Yaskawa INFORM job: DPRINT3D3.JBI

/JOB
//NAME DPRINT3D3
//POS
///NPOS 1003,0,0,0,0,0
///TOOL 9
///POSTYPE PULSE
///PULSE
C00000=29899,52059,-123343,60719,-118918,-94818,0
C00001=29890,52052,-123365,60727,-118907,-94823,0
C00002=29880,52046,-123386,60735,-118894,-94827,0
C00003=29870,52040,-123408,60743,-118882,-94832,0
C00004=29861,52034,-123430,60750,-118870,-94837,0
C00005=29851,52028,-123450,60758,-118858,-94842,0
C00006=29842,52022,-123472,60766,-118846,-94847,0
C00007=29832,52016,-123494,60774,-118834,-94852,0
C00008=29824,52011,-123510,60781,-118825,-94855,0
C00009=29816,52006,-123527,60788,-118815,-94859,0
C00010=29807,52001,-123543,60795,-118805,-94863,0
C00011=29799,51997,-123561,60802,-118795,-94866,0
C00012=29789,51992,-123577,60810,-118786,-94870,0
C00013=29780,51988,-123593,60818,-118777,-94872,0
C00014=29772,51983,-123609,60825,-118766,-94876,0
C00015=29762,51978,-123626,60833,-118757,-94879,0
C00016=29753,51974,-123642,60841,-118747,-94883,0
C00017=29744,51969,-123658,60849,-118738,-94886,0
C00018=29735,51964,-123674,60857,-118727,-94890,0
C00019=29726,51960,-123691,60865,-118718,-94893,0
C00020=29717,51955,-123707,60872,-118709,-94897,0
C00021=29708,51951,-123724,60880,-118699,-94900,0
C00022=29699,51946,-123740,60888,-118689,-94904,0
C00023=29690,51941,-123756,60896,-118680,-94907,0
C00024=29682,51937,-123770,60903,-118671,-94910,0
C00025=29674,51934,-123782,60911,-118663,-94912,0
C00026=29665,51930,-123796,60918,-118655,-94915,0
C00027=29657,51926,-123810,60926,-118647,-94918,0
C00028=29649,51922,-123824,60933,-118638,-94921,0
C00029=29640,51918,-123836,60941,-118630,-94924,0
C00030=29632,51915,-123850,60948,-118622,-94926,0
C00031=29624,51911,-123862,60956,-118614,-94929,0
C00032=29615,51908,-123874,60964,-118607,-94931,0
C00033=29611,51906,-123881,60968,-118602,-94932,0
C00034=29593,51903,-123889,60986,-118593,-94932,0
C00035=29559,51898,-123908,61022,-118574,-94933,0
C00036=29524,51893,-123925,61058,-118556,-94933,0
C00037=29489,51888,-123943,61094,-118537,-94934,0
C00038=29463,51884,-123955,61122,-118524,-94934,0
C00039=29436,51881,-123966,61150,-118510,-94933,0
C00040=29409,51878,-123977,61178,-118497,-94933,0
C00041=29384,51875,-123986,61204,-118486,-94932,0
C00042=29360,51873,-123994,61230,-118474,-94932,0
C00043=29335,51870,-124003,61256,-118463,-94931,0
C00044=29310,51868,-124011,61283,-118450,-94930,0
C00045=29285,51865,-124019,61309,-118439,-94929,0
C00046=29260,51863,-124028,61335,-118427,-94928,0
C00047=29238,51861,-124034,61359,-118418,-94928,0
C00048=29218,51859,-124040,61380,-118409,-94926,0
C00049=29198,51858,-124046,61402,-118401,-94925,0
C00050=29178,51856,-124050,61423,-118392,-94924,0
C00051=29158,51855,-124055,61445,-118384,-94923,0
C00052=29141,51853,-124059,61463,-118376,-94922,0
C00053=29134,51853,-124061,61471,-118373,-94921,0
C00054=29119,51858,-124043,61489,-118376,-94915,0
C00055=29105,51862,-124026,61506,-118378,-94908,0
C00056=29091,51867,-124010,61524,-118380,-94901,0
C00057=29077,51872,-123993,61542,-118383,-94894,0
C00058=29063,51876,-123975,61560,-118385,-94888,0
C00059=29049,51881,-123958,61577,-118387,-94881,0
C00060=29035,51886,-123941,61595,-118389,-94875,0
C00061=29021,51890,-123924,61613,-118392,-94868,0
C00062=29007,51895,-123907,61630,-118394,-94861,0
C00063=28992,51901,-123887,61650,-118397,-94853,0
C00064=28977,51906,-123866,61669,-118401,-94846,0
C00065=28962,51912,-123847,61688,-118404,-94838,0
C00066=28947,51917,-123826,61707,-118408,-94830,0
C00067=28931,51924,-123804,61727,-118411,-94822,0
C00068=28914,51931,-123779,61748,-118416,-94813,0
C00069=28898,51937,-123755,61770,-118420,-94803,0
C00070=28881,51944,-123730,61791,-118425,-94794,0
C00071=28865,51951,-123704,61813,-118430,-94785,0
C00072=28848,51958,-123680,61834,-118434,-94776,0
C00073=28832,51965,-123655,61855,-118439,-94766,0
C00074=28815,51972,-123631,61877,-118443,-94757,0
C00075=28799,51979,-123604,61898,-118449,-94748,0
C00076=28783,51987,-123578,61919,-118454,-94738,0
C00077=28767,51994,-123550,61940,-118460,-94728,0
C00078=28745,52005,-123510,61969,-118469,-94713,0
C00079=28723,52017,-123470,61999,-118478,-94699,0
C00080=28701,52028,-123428,62029,-118487,-94684,0
C00081=28679,52039,-123387,62058,-118496,-94670,0
C00082=28657,52051,-123347,62088,-118504,-94655,0
C00083=28633,52064,-123299,62120,-118517,-94639,0
C00084=28605,52082,-123237,62159,-118532,-94617,0
C00085=28573,52102,-123163,62204,-118550,-94592,0
C00086=28541,52123,-123088,62248,-118569,-94566,0
C00087=28512,52142,-123021,62289,-118587,-94543,0
C00088=28512,52148,-123000,62292,-118595,-94537,0
C00089=28511,52154,-122979,62295,-118603,-94531,0
C00090=28511,52160,-122960,62298,-118611,-94525,0
C00091=28511,52165,-122940,62300,-118618,-94520,0
C00092=28511,52171,-122918,62303,-118627,-94514,0
C00093=28512,52178,-122896,62305,-118637,-94507,0
C00094=28513,52185,-122872,62307,-118646,-94500,0
C00095=28514,52192,-122847,62310,-118656,-94494,0
C00096=28515,52199,-122823,62312,-118666,-94487,0
C00097=28515,52206,-122798,62314,-118677,-94480,0
C00098=28517,52213,-122773,62316,-118687,-94473,0
C00099=28518,52220,-122748,62318,-118697,-94466,0
C00100=28518,52227,-122724,62320,-118707,-94459,0
C00101=28519,52234,-122699,62322,-118717,-94452,0
C00102=28520,52241,-122675,62325,-118727,-94445,0
C00103=28521,52248,-122649,62327,-118738,-94438,0
C00104=28522,52255,-122624,62329,-118748,-94431,0
C00105=28544,52343,-122318,62346,-118877,-94346,0
C00106=28565,52431,-122013,62363,-119005,-94261,0
C00107=22726,60437,-97506,72380,-124352,-86432,0
C00108=22603,60494,-97345,72531,-124324,-86367,0
C00109=22480,60552,-97184,72683,-124295,-86302,0
C00110=22469,60557,-97168,72696,-124293,-86296,0
C00111=22459,60563,-97152,72710,-124290,-86289,0
C00112=22448,60569,-97136,72724,-124288,-86283,0
C00113=22437,60574,-97120,72737,-124286,-86277,0
C00114=22427,60580,-97104,72751,-124285,-86271,0
C00115=22416,60586,-97088,72764,-124282,-86264,0
C00116=22405,60591,-97072,72778,-124280,-86258,0
C00117=22394,60597,-97057,72791,-124278,-86252,0
C00118=22384,60603,-97041,72805,-124275,-86246,0
C00119=22373,60608,-97025,72818,-124273,-86239,0
C00120=22362,60614,-97009,72832,-124272,-86233,0
C00121=22352,60619,-96994,72844,-124270,-86227,0
C00122=22344,60625,-96980,72855,-124269,-86222,0
C00123=22335,60630,-96965,72866,-124267,-86217,0
C00124=22327,60635,-96951,72877,-124266,-86211,0
C00125=22318,60640,-96936,72888,-124265,-86206,0
C00126=22310,60645,-96921,72900,-124264,-86200,0
C00127=22302,60651,-96905,72911,-124263,-86194,0
C00128=22293,60657,-96890,72922,-124263,-86188,0
C00129=22285,60662,-96875,72933,-124262,-86182,0
C00130=22277,60668,-96859,72944,-124260,-86177,0
C00131=22268,60673,-96843,72955,-124259,-86171,0
C00132=22260,60679,-96828,72966,-124259,-86166,0
C00133=22251,60684,-96812,72977,-124258,-86160,0
C00134=22225,60745,-96644,73033,-124287,-86108,0
C00135=22211,60785,-96532,73066,-124309,-86074,0
C00136=22198,60827,-96416,73100,-124332,-86039,0
C00137=22185,60869,-96300,73134,-124354,-86004,0
C00138=22179,60891,-96239,73150,-124367,-85986,0
C00139=22173,60913,-96177,73167,-124380,-85967,0
C00140=22169,60935,-96117,73181,-124393,-85950,0
C00141=22165,60956,-96059,73196,-124406,-85932,0
C00142=22161,60977,-96000,73210,-124419,-85915,0
C00143=22157,60998,-95940,73225,-124432,-85897,0
C00144=22153,61020,-95881,73239,-124446,-85880,0
C00145=22150,61038,-95832,73250,-124457,-85866,0
C00146=22148,61055,-95783,73261,-124468,-85852,0
C00147=22145,61073,-95734,73272,-124480,-85837,0
C00148=22144,61089,-95691,73281,-124490,-85825,0
C00149=22143,61104,-95648,73290,-124501,-85813,0
C00150=22142,61120,-95605,73299,-124511,-85800,0
C00151=22141,61135,-95563,73307,-124521,-85788,0
C00152=22139,61151,-95520,73316,-124532,-85776,0
C00153=22138,61166,-95477,73325,-124543,-85763,0
C00154=22137,61182,-95434,73334,-124554,-85751,0
C00155=22137,61195,-95397,73340,-124563,-85740,0
C00156=22137,61209,-95359,73347,-124572,-85730,0
C00157=22136,61222,-95322,73354,-124582,-85719,0
C00158=22136,61236,-95285,73361,-124591,-85708,0
C00159=22136,61249,-95248,73368,-124601,-85698,0
C00160=22136,61261,-95215,73373,-124610,-85689,0
C00161=22137,61273,-95183,73378,-124619,-85679,0
C00162=22137,61285,-95150,73384,-124627,-85671,0
C00163=22138,61297,-95117,73389,-124636,-85661,0
C00164=22138,61309,-95085,73394,-124645,-85652,0
C00165=22139,61320,-95052,73400,-124653,-85643,0
C00166=22139,61332,-95019,73405,-124663,-85633,0
C00167=22139,61344,-94987,73411,-124672,-85624,0
C00168=22153,61355,-94956,73403,-124687,-85618,0
C00169=22165,61365,-94930,73395,-124702,-85613,0
C00170=22178,61374,-94904,73387,-124717,-85607,0
C00171=22190,61384,-94878,73379,-124730,-85602,0
C00172=22203,61394,-94852,73372,-124745,-85596,0
C00173=22215,61403,-94825,73364,-124759,-85591,0
C00174=22231,61414,-94797,73354,-124776,-85585,0
C00175=22246,61424,-94768,73344,-124794,-85580,0
C00176=22261,61435,-94739,73334,-124811,-85574,0
C00177=22277,61446,-94710,73324,-124827,-85568,0
C00178=22292,61456,-94681,73314,-124844,-85563,0
C00179=22307,61467,-94651,73304,-124861,-85557,0
C00180=22326,61479,-94619,73290,-124882,-85551,0
C00181=22345,61491,-94587,73278,-124902,-85545,0
C00182=22364,61502,-94554,73265,-124922,-85539,0
C00183=22388,61516,-94517,73248,-124947,-85532,0
C00184=22412,61529,-94481,73231,-124971,-85526,0
C00185=22421,61530,-94478,73222,-124976,-85527,0
C00186=22431,61531,-94476,73213,-124983,-85527,0
C00187=22440,61532,-94473,73204,-124989,-85528,0
C00188=22449,61533,-94470,73195,-124996,-85529,0
C00189=22458,61535,-94467,73187,-125002,-85530,0
C00190=22468,61535,-94465,73178,-125009,-85531,0
C00191=22477,61537,-94462,73169,-125015,-85531,0
C00192=22487,61537,-94460,73160,-125021,-85532,0
C00193=22497,61538,-94459,73150,-125028,-85534,0
C00194=22507,61539,-94457,73141,-125034,-85535,0
C00195=22517,61539,-94455,73131,-125041,-85536,0
C00196=22526,61540,-94453,73122,-125048,-85537,0
C00197=22536,61541,-94452,73112,-125055,-85538,0
C00198=38402,60566,-97394,77280,-121677,-85721,0
C00199=38418,60624,-97233,77289,-121724,-85676,0
C00200=38452,60740,-96909,77308,-121819,-85588,0
C00201=38470,60804,-96733,77318,-121870,-85539,0
C00202=38473,60814,-96704,77319,-121879,-85531,0
C00203=38477,60825,-96675,77320,-121887,-85524,0
C00204=38480,60835,-96646,77321,-121897,-85516,0
C00205=38484,60846,-96617,77322,-121906,-85508,0
C00206=38488,60856,-96588,77323,-121914,-85500,0
C00207=38491,60866,-96560,77324,-121923,-85492,0
C00208=38495,60877,-96531,77326,-121932,-85484,0
C00209=38498,60887,-96501,77327,-121941,-85476,0
C00210=38502,60898,-96473,77328,-121950,-85469,0
C00211=38505,60908,-96444,77329,-121959,-85461,0
C00212=38509,60919,-96415,77330,-121968,-85453,0
C00213=38512,60927,-96391,77330,-121975,-85447,0
C00214=38516,60936,-96368,77331,-121983,-85440,0
C00215=38519,60944,-96344,77331,-121990,-85434,0
C00216=38523,60953,-96320,77332,-121998,-85427,0
C00217=38527,60961,-96297,77331,-122006,-85421,0
C00218=38531,60970,-96273,77331,-122013,-85415,0
C00219=38534,60978,-96250,77331,-122021,-85409,0
C00220=38538,60987,-96226,77331,-122029,-85402,0
C00221=38542,60996,-96203,77331,-122037,-85396,0
C00222=38546,61004,-96179,77331,-122045,-85390,0
C00223=38550,61013,-96156,77331,-122053,-85384,0
C00224=38554,61021,-96132,77331,-122060,-85378,0
C00225=38556,61025,-96120,77330,-122064,-85375,0
C00226=38617,61064,-96014,77289,-122127,-85352,0
C00227=38658,61088,-95950,77259,-122166,-85340,0
C00228=38700,61111,-95887,77227,-122207,-85328,0
C00229=38743,61134,-95824,77196,-122248,-85315,0
C00230=38766,61145,-95793,77178,-122269,-85310,0
C00231=38789,61157,-95762,77161,-122291,-85304,0
C00232=38812,61166,-95736,77143,-122310,-85300,0
C00233=38834,61176,-95710,77125,-122330,-85295,0
C00234=38856,61185,-95684,77108,-122351,-85291,0
C00235=38879,61195,-95657,77090,-122370,-85286,0
C00236=38901,61205,-95631,77073,-122390,-85282,0
C00237=38920,61212,-95611,77058,-122406,-85279,0
C00238=38938,61219,-95592,77042,-122422,-85276,0
C00239=38957,61226,-95573,77027,-122438,-85273,0
C00240=38974,61232,-95557,77014,-122452,-85271,0
C00241=38990,61238,-95542,77000,-122466,-85270,0
C00242=39007,61243,-95527,76986,-122479,-85267,0
C00243=39024,61249,-95512,76972,-122493,-85266,0
C00244=39040,61254,-95497,76958,-122507,-85264,0
C00245=39057,61260,-95482,76945,-122521,-85261,0
C00246=39073,61265,-95467,76931,-122534,-85260,0
C00247=39088,61270,-95456,76918,-122546,-85259,0
C00248=39103,61274,-95445,76906,-122557,-85257,0
C00249=39117,61278,-95434,76894,-122570,-85256,0
C00250=39132,61282,-95422,76881,-122582,-85255,0
C00251=39146,61286,-95411,76869,-122593,-85254,0
C00252=39159,61289,-95403,76857,-122603,-85253,0
C00253=39172,61292,-95395,76846,-122613,-85253,0
C00254=39185,61296,-95386,76835,-122623,-85253,0
C00255=39198,61299,-95378,76824,-122633,-85252,0
C00256=39211,61302,-95370,76812,-122642,-85252,0
C00257=39224,61305,-95361,76801,-122653,-85251,0
C00258=39237,61308,-95353,76790,-122663,-85250,0
C00259=39250,61311,-95344,76779,-122672,-85250,0
C00260=39255,61309,-95352,76772,-122675,-85253,0
C00261=39266,61303,-95367,76760,-122677,-85259,0
C00262=39280,61295,-95389,76742,-122680,-85267,0
C00263=39293,61288,-95410,76725,-122684,-85275,0
C00264=39307,61280,-95432,76708,-122687,-85284,0
C00265=39321,61272,-95454,76691,-122691,-85292,0
C00266=39335,61264,-95476,76674,-122694,-85300,0
C00267=39351,61254,-95503,76654,-122698,-85310,0
C00268=39366,61244,-95531,76634,-122701,-85320,0
C00269=39382,61234,-95558,76614,-122705,-85331,0
C00270=39398,61225,-95586,76594,-122708,-85340,0
C00271=39414,61215,-95614,76574,-122711,-85351,0
C00272=39430,61205,-95641,76554,-122714,-85361,0
C00273=39448,61192,-95676,76530,-122717,-85374,0
C00274=39466,61180,-95711,76507,-122721,-85387,0
C00275=39484,61167,-95746,76483,-122723,-85400,0
C00276=39506,61151,-95791,76455,-122725,-85415,0
C00277=39527,61135,-95836,76427,-122728,-85432,0
C00278=39530,61127,-95858,76420,-122725,-85438,0
C00279=39534,61120,-95879,76413,-122723,-85444,0
C00280=39538,61112,-95899,76406,-122719,-85451,0
C00281=39542,61105,-95920,76398,-122717,-85458,0
C00282=39545,61097,-95941,76391,-122715,-85464,0
C00283=39549,61089,-95962,76384,-122711,-85471,0
C00284=39553,61082,-95983,76377,-122709,-85477,0
C00285=39556,61074,-96006,76370,-122706,-85484,0
C00286=39560,61066,-96028,76363,-122703,-85491,0
C00287=39563,61058,-96051,76356,-122700,-85498,0
C00288=39567,61050,-96073,76348,-122696,-85505,0
C00289=39571,61041,-96096,76341,-122693,-85512,0
C00290=39574,61033,-96118,76334,-122691,-85519,0
C00291=40253,57939,-104914,74266,-120876,-88158,0
C00292=39352,58001,-104714,75214,-120443,-87977,0
C00293=39289,57986,-104756,75273,-120398,-87981,0
C00294=38619,57932,-104903,75932,-119998,-87936,0
C00295=37942,57980,-104749,76638,-119667,-87804,0
C00296=37297,58130,-104299,77353,-119421,-87590,0
C00297=37222,58161,-104207,77441,-119401,-87554,0
C00298=36275,57663,-105643,78197,-118546,-87864,0
C00299=41043,57280,-106870,73160,-120764,-88836,0
C00300=41858,56647,-108775,72029,-120639,-89503,0
C00301=35258,57163,-107098,79033,-117663,-88181,0
C00302=34216,56686,-108501,79913,-116799,-88491,0
C00303=42701,56041,-110631,70871,-120503,-90160,0
C00304=43572,55460,-112438,69686,-120353,-90807,0
C00305=33148,56231,-109853,80834,-115950,-88792,0
C00306=32056,55798,-111153,81799,-115118,-89085,0
C00307=44472,54905,-114198,68471,-120191,-91442,0
C00308=45402,54374,-115911,67227,-120017,-92067,0
C00309=30938,55387,-112402,82805,-114303,-89372,0
C00310=30073,55089,-113315,83596,-113696,-89584,0
C00311=30084,55047,-113445,83573,-113676,-89626,0
C00312=30076,54952,-113743,83553,-113615,-89719,0
C00313=46130,53866,-117579,66205,-119735,-92649,0
C00314=46001,53590,-118484,66218,-119365,-92894,0
C00315=45984,53367,-119225,66135,-119095,-93108,0
C00316=25619,60155,-98330,69289,-125787,-87153,0
C00317=25520,59915,-99002,69267,-125531,-87324,0
C00318=25252,59544,-100046,69355,-125071,-87569,0
C00319=46086,52886,-120853,65807,-118548,-93596,0
C00320=46100,52846,-120989,65774,-118503,-93638,0
C00321=46138,52799,-121152,65710,-118458,-93690,0
C00322=45305,52415,-122459,66450,-117684,-93972,0
C00323=25512,58771,-102250,68697,-124545,-88230,0
C00324=26027,57961,-104598,67753,-124084,-88973,0
C00325=44250,51964,-124020,67407,-116754,-94317,0
C00326=36507,55621,-111785,55133,-126158,-92810,0
C00327=26561,57182,-106893,66801,-123611,-89703,0
C00328=27117,56433,-109139,65839,-123127,-90421,0
C00329=35436,55163,-113183,56093,-125149,-92963,0
C00330=34338,54728,-114530,57095,-124159,-93114,0
C00331=27695,55714,-111338,64867,-122633,-91128,0
C00332=28295,55023,-113491,63881,-122127,-91823,0
C00333=33211,54314,-115828,58137,-123193,-93261,0
C00334=32057,53921,-117076,59221,-122246,-93405,0
C00335=31078,54046,-116653,60363,-122047,-93134,0
C00336=31078,53985,-116676,60373,-122074,-93115,0
C00337=46650,54077,-116730,65775,-120275,-92451,0
C00338=46377,53734,-117841,65913,-119772,-92732,0
C00339=46298,53541,-118474,65910,-119517,-92905,0
C00340=46256,53321,-119205,65855,-119239,-93111,0
C00341=46316,53032,-120175,65658,-118912,-93401,0
C00342=46494,52760,-121103,65341,-118639,-93694,0
C00343=46678,52606,-121638,65070,-118508,-93874,0
C00344=31635,53384,-118654,59466,-121484,-93741,0
C00345=31072,53603,-117924,60193,-121574,-93455,0
C00346=30731,53690,-117631,60612,-121562,-93322,0
C00347=30325,53768,-117369,61095,-121513,-93187,0
C00348=29755,53817,-117197,61746,-121361,-93053,0
C00349=29175,53810,-117209,62378,-121132,-92969,0
C00350=28816,53770,-117336,62751,-120945,-92950,0
C00351=24539,59459,-100146,70086,-124670,-87452,0
C00352=24731,59594,-99769,69956,-124888,-87378,0
C00353=25015,59895,-98924,69816,-125295,-87190,0
C00354=25218,60240,-97961,69783,-125692,-86956,0
C00355=25335,60616,-96916,69857,-126065,-86685,0
C00356=25361,61009,-95827,70034,-126396,-86386,0
C00357=29506,55205,-112783,84233,-113529,-89344,0
C00358=37736,58857,-102075,77244,-120213,-86968,0
C00359=37945,58742,-102408,76986,-120253,-87092,0
C00360=38379,58595,-102839,76487,-120395,-87275,0
C00361=38845,58519,-103067,75985,-120599,-87403,0
C00362=39320,58515,-103088,75502,-120859,-87473,0
C00363=39792,58584,-102900,75054,-121169,-87483,0
C00364=40036,58660,-102685,74841,-121359,-87455,0
C00365=46580,54114,-116609,65869,-120289,-92406,0
C00366=47912,54121,-116622,64422,-120819,-92601,0
C00367=47637,53970,-117105,64650,-120534,-92698,0
C00368=47420,53795,-117671,64805,-120243,-92829,0
C00369=47270,53603,-118298,64879,-119957,-92987,0
C00370=47224,53482,-118695,64873,-119794,-93095,0
C00371=47201,53334,-119186,64830,-119605,-93233,0
C00372=47248,53136,-119851,64687,-119378,-93430,0
C00373=47376,52949,-120486,64461,-119189,-93631,0
C00374=47579,52781,-121062,64161,-119047,-93824,0
C00375=47741,52695,-121362,63943,-118990,-93932,0
C00376=47974,52598,-121700,63644,-118944,-94061,0
C00377=31349,52761,-120741,59484,-120523,-94269,0
C00378=31148,52930,-120165,59786,-120690,-94082,0
C00379=30885,53077,-119663,60147,-120803,-93904,0
C00380=30567,53199,-119249,60557,-120854,-93743,0
C00381=30351,53253,-119065,60820,-120850,-93660,0
C00382=30075,53305,-118888,61149,-120819,-93570,0
C00383=29678,53339,-118769,61602,-120719,-93478,0
C00384=29274,53334,-118778,62043,-120565,-93421,0
C00385=28879,53290,-118913,62456,-120365,-93402,0
C00386=28654,53243,-119069,62680,-120221,-93413,0
C00387=28385,53168,-119313,62940,-120026,-93444,0
C00388=23547,59693,-99475,71219,-124304,-87099,0
C00389=23788,59787,-99213,71019,-124516,-87064,0
C00390=24041,59943,-98776,70839,-124785,-86984,0
C00391=24084,59984,-98662,70815,-124842,-86959,0
C00392=24158,60037,-98516,70765,-124926,-86930,0
C00393=24348,60239,-97953,70673,-125196,-86804,0
C00394=24486,60470,-97312,70649,-125458,-86648,0
C00395=24567,60721,-96615,70694,-125703,-86467,0
C00396=24589,60983,-95890,70807,-125921,-86267,0
C00397=24551,61249,-95155,70982,-126106,-86055,0
C00398=24417,61602,-94184,71298,-126296,-85760,0
C00399=37795,59676,-99749,77530,-120789,-86297,0
C00400=37965,59511,-100218,77291,-120780,-86456,0
C00401=38212,59353,-100672,76977,-120818,-86621,0
C00402=38272,59329,-100741,76908,-120836,-86649,0
C00403=38352,59284,-100870,76809,-120852,-86698,0
C00404=38638,59185,-101157,76480,-120949,-86819,0
C00405=38944,59134,-101309,76151,-121088,-86905,0
C00406=39256,59131,-101323,75836,-121262,-86952,0
C00407=39567,59177,-101197,75544,-121471,-86958,0
C00408=39859,59272,-100935,75291,-121704,-86924,0
C00409=40225,59466,-100391,75010,-122050,-86819,0
C00410=47839,54157,-116505,64518,-120833,-92557,0
C00411=48074,53235,-119541,63828,-119801,-93454,0
C00412=48152,53124,-119916,63691,-119688,-93572,0
C00413=48274,53024,-120256,63510,-119603,-93686,0
C00414=48351,52983,-120396,63407,-119578,-93737,0
C00415=48477,52930,-120580,63244,-119552,-93806,0
C00416=48685,52874,-120776,62989,-119551,-93891,0
C00417=48910,52840,-120899,62724,-119585,-93957,0
C00418=49522,52810,-121018,62036,-119754,-94075,0
C00419=30592,52097,-123019,60009,-119319,-94794,0
C00420=30654,52388,-122008,60076,-119760,-94520,0
C00421=30630,52493,-121643,60152,-119903,-94415,0
C00422=30560,52596,-121288,60278,-120025,-94307,0
C00423=30446,52693,-120953,60449,-120121,-94198,0
C00424=30293,52779,-120659,60659,-120188,-94094,0
C00425=30105,52850,-120414,60900,-120220,-93999,0
C00426=30003,52875,-120328,61025,-120219,-93960,0
C00427=29845,52904,-120228,61212,-120203,-93909,0
C00428=29607,52923,-120157,61483,-120145,-93855,0
C00429=29365,52920,-120163,61749,-120056,-93822,0
C00430=29127,52895,-120243,61998,-119937,-93811,0
C00431=29021,52873,-120317,62105,-119871,-93817,0
C00432=28873,52833,-120450,62248,-119765,-93834,0
C00433=28689,52757,-120703,62415,-119601,-93880,0
C00434=28541,52668,-121003,62537,-119429,-93945,0
C00435=28257,52411,-121881,62731,-118986,-94156,0
C00436=22514,60235,-97942,72532,-124133,-86498,0
C00437=22908,60179,-98103,72106,-124319,-86607,0
C00438=23091,60184,-98090,71924,-124429,-86633,0
C00439=23266,60220,-97993,71764,-124558,-86634,0
C00440=23426,60283,-97817,71633,-124699,-86611,0
C00441=23566,60371,-97574,71534,-124849,-86566,0
C00442=23596,60400,-97495,71518,-124888,-86549,0
C00443=23656,60442,-97377,71479,-124956,-86525,0
C00444=23762,60555,-97066,71428,-125105,-86456,0
C00445=23839,60683,-96711,71414,-125249,-86369,0
C00446=23885,60822,-96326,71437,-125383,-86268,0
C00447=23899,60967,-95925,71496,-125503,-86158,0
C00448=23880,61113,-95522,71589,-125603,-86042,0
C00449=23828,61256,-95128,71715,-125680,-85922,0
C00450=23750,61381,-94782,71856,-125727,-85812,0
C00451=23723,61410,-94703,71898,-125733,-85785,0
C00452=23681,61470,-94537,71971,-125752,-85731,0
C00453=23564,61582,-94229,72145,-125764,-85624,0
C00454=23225,61801,-93628,72594,-125718,-85397,0
C00455=38177,60645,-97044,77569,-121639,-85564,0
C00456=38213,60309,-97979,77388,-121446,-85839,0
C00457=38265,60164,-98388,77273,-121384,-85965,0
C00458=38350,60032,-98757,77132,-121349,-86084,0
C00459=38464,59921,-99072,76971,-121343,-86190,0
C00460=38601,59832,-99324,76797,-121365,-86282,0
C00461=38642,59816,-99372,76749,-121377,-86302,0
C00462=38706,59779,-99476,76669,-121391,-86341,0
C00463=38863,59724,-99635,76489,-121445,-86409,0
C00464=39030,59695,-99719,76309,-121523,-86456,0
C00465=39200,59694,-99727,76139,-121621,-86482,0
C00466=39370,59720,-99657,75981,-121737,-86485,0
C00467=39530,59772,-99512,75844,-121866,-86466,0
C00468=39673,59849,-99298,75736,-122002,-86425,0
C00469=39796,59948,-99024,75658,-122141,-86363,0
C00470=39820,59977,-98940,75647,-122176,-86343,0
C00471=39875,60027,-98802,75614,-122243,-86311,0
C00472=39966,60153,-98451,75581,-122383,-86222,0
C00473=40107,60492,-97507,75594,-122699,-85972,0
C00474=49430,53986,-117100,62696,-121237,-92960,0
C00475=48830,53910,-117331,63318,-120918,-92936,0
C00476=48628,53862,-117483,63517,-120782,-92949,0
C00477=48443,53793,-117702,63686,-120629,-92984,0
C00478=48285,53707,-117982,63819,-120464,-93041,0
C00479=48159,53605,-118314,63908,-120292,-93117,0
C00480=48073,53493,-118684,63949,-120121,-93210,0
C00481=48053,53436,-118870,63945,-120044,-93260,0
C00482=48042,53353,-119147,63918,-119936,-93338,0
C00483=48061,53285,-119373,63866,-119858,-93405,0
C00484=47899,53152,-119813,63982,-119633,-93508,0
C00485=49346,53759,-117839,62680,-120923,-93155,0
C00486=49500,53752,-117865,62507,-120970,-93185,0
C00487=49654,53746,-117892,62335,-121020,-93215,0
C00488=49669,53745,-117895,62318,-121023,-93219,0
C00489=49684,53744,-117899,62301,-121028,-93222,0
C00490=49699,53742,-117905,62283,-121031,-93226,0
C00491=49715,53741,-117910,62265,-121036,-93230,0
C00492=49731,53739,-117915,62247,-121039,-93233,0
C00493=49747,53738,-117921,62229,-121044,-93237,0
C00494=49762,53736,-117926,62211,-121047,-93241,0
C00495=49778,53735,-117931,62193,-121051,-93245,0
C00496=49794,53733,-117937,62175,-121055,-93249,0
C00497=49809,53732,-117941,62157,-121059,-93252,0
C00498=49823,53731,-117947,62141,-121062,-93256,0
C00499=49836,53729,-117952,62126,-121065,-93259,0
C00500=49849,53728,-117957,62112,-121068,-93263,0
C00501=49861,53726,-117963,62097,-121070,-93266,0
C00502=49874,53724,-117969,62082,-121073,-93270,0
C00503=49887,53722,-117976,62067,-121075,-93273,0
C00504=49900,53720,-117982,62052,-121077,-93277,0
C00505=49912,53719,-117988,62037,-121080,-93281,0
C00506=49925,53717,-117994,62022,-121082,-93284,0
C00507=49938,53715,-118001,62007,-121084,-93288,0
C00508=49951,53713,-118007,61992,-121087,-93292,0
C00509=49964,53711,-118014,61978,-121089,-93295,0
C00510=49976,53710,-118021,61962,-121091,-93299,0
C00511=49989,53708,-118026,61948,-121093,-93303,0
C00512=50002,53706,-118033,61933,-121096,-93307,0
C00513=50014,53704,-118039,61918,-121098,-93310,0
C00514=50025,53702,-118046,61905,-121100,-93314,0
C00515=50037,53700,-118053,61892,-121101,-93317,0
C00516=50048,53698,-118060,61878,-121103,-93321,0
C00517=50059,53696,-118067,61865,-121105,-93324,0
C00518=50071,53694,-118072,61851,-121106,-93328,0
C00519=50082,53692,-118079,61838,-121108,-93332,0
C00520=50091,53690,-118086,61827,-121110,-93335,0
C00521=50100,53689,-118092,61816,-121110,-93338,0
C00522=50109,53687,-118099,61805,-121111,-93341,0
C00523=50137,53671,-118153,61767,-121100,-93360,0
C00524=50164,53654,-118207,61729,-121089,-93379,0
C00525=50188,53640,-118254,61697,-121080,-93396,0
C00526=50206,53628,-118295,61670,-121070,-93410,0
C00527=50225,53616,-118335,61643,-121061,-93425,0
C00528=50241,53605,-118372,61621,-121053,-93437,0
C00529=50256,53594,-118409,61599,-121044,-93449,0
C00530=50271,53583,-118446,61577,-121036,-93462,0
C00531=50286,53572,-118483,61555,-121027,-93474,0
C00532=50302,53561,-118518,61533,-121018,-93487,0
C00533=50314,53552,-118550,61515,-121010,-93497,0
C00534=50326,53542,-118583,61497,-121001,-93508,0
C00535=50338,53532,-118615,61479,-120993,-93519,0
C00536=50350,53523,-118646,61461,-120985,-93529,0
C00537=50359,53514,-118674,61447,-120979,-93538,0
C00538=50369,53506,-118703,61432,-120970,-93548,0
C00539=50379,53497,-118732,61417,-120962,-93558,0
C00540=50388,53489,-118761,61402,-120956,-93567,0
C00541=50398,53480,-118788,61388,-120947,-93576,0
C00542=50408,53472,-118817,61373,-120939,-93585,0
C00543=50417,53463,-118846,61358,-120931,-93595,0
C00544=50426,53456,-118872,61345,-120924,-93603,0
C00545=50434,53448,-118899,61332,-120918,-93612,0
C00546=50443,53440,-118924,61319,-120911,-93620,0
C00547=50440,53436,-118938,61320,-120904,-93624,0
C00548=50434,53427,-118966,61323,-120890,-93631,0
C00549=50428,53419,-118994,61325,-120877,-93638,0
C00550=50421,53410,-119024,61328,-120864,-93645,0
C00551=50414,53401,-119054,61332,-120849,-93652,0
C00552=50407,53391,-119085,61335,-120834,-93660,0
C00553=50400,53382,-119115,61338,-120819,-93667,0
C00554=50393,53373,-119146,61342,-120805,-93675,0
C00555=50386,53364,-119175,61345,-120790,-93682,0
C00556=50379,53355,-119207,61349,-120775,-93689,0
C00557=50370,53345,-119239,61353,-120759,-93697,0
C00558=50361,53334,-119273,61358,-120743,-93706,0
C00559=50352,53324,-119308,61363,-120726,-93714,0
C00560=50343,53314,-119342,61369,-120708,-93722,0
C00561=50332,53302,-119379,61375,-120690,-93731,0
C00562=50320,53290,-119419,61383,-120669,-93740,0
C00563=50308,53279,-119458,61390,-120650,-93750,0
C00564=50296,53267,-119498,61398,-120629,-93759,0
C00565=50284,53255,-119537,61406,-120610,-93768,0
C00566=50270,53242,-119580,61415,-120588,-93777,0
C00567=50254,53228,-119625,61426,-120565,-93788,0
C00568=50239,53215,-119670,61436,-120542,-93798,0
C00569=50218,53199,-119724,61452,-120512,-93811,0
C00570=50203,53187,-119763,61462,-120491,-93819,0
C00571=50190,53175,-119802,61472,-120472,-93828,0
C00572=50170,53159,-119853,61486,-120444,-93840,0
C00573=50151,53144,-119904,61500,-120417,-93851,0
C00574=50141,53137,-119927,61508,-120404,-93856,0
C00575=50136,53136,-119932,61512,-120400,-93856,0
C00576=50125,53133,-119941,61523,-120394,-93858,0
C00577=50115,53130,-119950,61533,-120386,-93859,0
C00578=50105,53128,-119959,61543,-120379,-93860,0
C00579=50095,53125,-119967,61553,-120372,-93861,0
C00580=50084,53122,-119976,61563,-120364,-93862,0
C00581=50074,53119,-119986,61573,-120357,-93863,0
C00582=50064,53117,-119995,61583,-120350,-93864,0
C00583=50053,53114,-120004,61593,-120343,-93865,0
C00584=50043,53111,-120013,61603,-120335,-93866,0
C00585=50033,53108,-120022,61613,-120328,-93867,0
C00586=50021,53106,-120030,61624,-120320,-93868,0
C00587=50010,53103,-120040,61635,-120313,-93869,0
C00588=49999,53100,-120049,61647,-120305,-93870,0
C00589=49988,53098,-120057,61658,-120298,-93870,0
C00590=49976,53095,-120066,61669,-120290,-93871,0
C00591=49964,53092,-120074,61682,-120282,-93872,0
C00592=49951,53089,-120083,61695,-120274,-93873,0
C00593=49938,53087,-120091,61707,-120266,-93873,0
C00594=49925,53084,-120101,61720,-120259,-93874,0
C00595=49913,53081,-120109,61733,-120251,-93874,0
C00596=49900,53079,-120118,61746,-120243,-93875,0
C00597=49887,53076,-120126,61759,-120235,-93876,0
C00598=49874,53074,-120135,61771,-120227,-93876,0
C00599=49861,53071,-120143,61784,-120219,-93877,0
C00600=49849,53068,-120151,61797,-120211,-93877,0
C00601=49836,53066,-120160,61810,-120203,-93878,0
C00602=49752,53050,-120209,61895,-120153,-93880,0
C00603=49598,53023,-120298,62053,-120064,-93883,0
C00604=49443,52996,-120386,62210,-119974,-93885,0
C00605=30185,52197,-122662,60505,-119333,-94639,0
C00606=30117,52131,-122893,60550,-119215,-94694,0
C00607=30049,52065,-123123,60595,-119097,-94749,0
C00608=30041,52059,-123145,60601,-119086,-94755,0
C00609=30034,52052,-123168,60606,-119074,-94760,0
C00610=30025,52046,-123189,60613,-119062,-94765,0
C00611=30017,52040,-123211,60619,-119050,-94770,0
C00612=30009,52033,-123233,60625,-119039,-94775,0
C00613=30000,52027,-123255,60632,-119026,-94780,0
C00614=29992,52021,-123278,60638,-119015,-94785,0
C00615=29983,52014,-123300,60645,-119003,-94790,0
C00616=29975,52008,-123322,60651,-118990,-94795,0
C00617=29966,52002,-123343,60657,-118979,-94800,0
C00618=29958,51996,-123365,60664,-118966,-94806,0
C00619=29950,51990,-123384,60670,-118956,-94810,0
C00620=29942,51985,-123403,60677,-118947,-94814,0
C00621=29934,51980,-123420,60683,-118936,-94818,0
C00622=29926,51975,-123439,60689,-118926,-94822,0
C00623=29918,51970,-123456,60696,-118917,-94825,0
C00624=29910,51965,-123473,60703,-118907,-94829,0
C00625=29902,51960,-123489,60710,-118897,-94833,0
C00626=29894,51955,-123507,60716,-118887,-94837,0
C00627=29885,51950,-123524,60723,-118878,-94841,0
C00628=29877,51946,-123541,60730,-118869,-94844,0
C00629=29869,51941,-123558,60736,-118858,-94848,0
C00630=29861,51936,-123574,60743,-118849,-94852,0
C00631=29853,51931,-123592,60750,-118839,-94856,0
C00632=29845,51926,-123609,60757,-118830,-94859,0
C00633=29837,51922,-123626,60763,-118820,-94863,0
C00634=29829,51917,-123640,60770,-118811,-94866,0
C00635=29821,51913,-123655,60777,-118802,-94869,0
C00636=29813,51909,-123670,60784,-118794,-94872,0
C00637=29805,51905,-123685,60790,-118785,-94875,0
C00638=29798,51901,-123700,60797,-118777,-94879,0
C00639=29790,51896,-123715,60804,-118768,-94882,0
C00640=29782,51893,-123727,60811,-118759,-94885,0
C00641=29775,51889,-123740,60817,-118753,-94887,0
C00642=29768,51886,-123751,60823,-118746,-94889,0
C00643=29765,51884,-123757,60826,-118742,-94890,0
C00644=29744,51880,-123770,60848,-118730,-94892,0
C00645=29702,51873,-123794,60891,-118707,-94893,0
C00646=29660,51866,-123818,60934,-118682,-94894,0
C00647=29628,51862,-123833,60967,-118666,-94894,0
C00648=29597,51858,-123849,60999,-118649,-94894,0
C00649=29567,51854,-123862,61030,-118634,-94894,0
C00650=29540,51850,-123873,61059,-118620,-94894,0
C00651=29512,51847,-123885,61088,-118608,-94893,0
C00652=29485,51844,-123895,61117,-118594,-94893,0
C00653=29457,51841,-123907,61146,-118580,-94893,0
C00654=29432,51838,-123916,61173,-118569,-94892,0
C00655=29409,51835,-123924,61197,-118557,-94891,0
C00656=29385,51833,-123931,61222,-118547,-94890,0
C00657=29362,51831,-123938,61247,-118537,-94889,0
C00658=29340,51829,-123944,61270,-118526,-94888,0
C00659=29320,51828,-123949,61292,-118518,-94887,0
C00660=29300,51826,-123954,61313,-118509,-94886,0
C00661=29280,51825,-123959,61335,-118501,-94885,0
C00662=29259,51823,-123964,61357,-118492,-94883,0
C00663=29239,51822,-123969,61379,-118484,-94882,0
C00664=29219,51820,-123973,61400,-118474,-94881,0
C00665=29199,51819,-123978,61421,-118466,-94879,0
C00666=29181,51818,-123981,61441,-118460,-94878,0
C00667=29162,51817,-123986,61461,-118452,-94877,0
C00668=29153,51816,-123987,61471,-118448,-94876,0
C00669=29138,51821,-123969,61489,-118450,-94869,0
C00670=29124,51826,-123950,61508,-118454,-94862,0
C00671=29110,51832,-123932,61526,-118456,-94854,0
C00672=29094,51837,-123910,61545,-118460,-94846,0
C00673=29079,51843,-123889,61565,-118463,-94838,0
C00674=29063,51849,-123867,61585,-118468,-94831,0
C00675=29048,51855,-123847,61605,-118471,-94823,0
C00676=29033,51861,-123826,61624,-118474,-94814,0
C00677=29017,51867,-123804,61644,-118478,-94806,0
C00678=29002,51873,-123784,61664,-118481,-94798,0
C00679=28985,51880,-123757,61686,-118486,-94789,0
C00680=28968,51887,-123732,61707,-118491,-94779,0
C00681=28951,51894,-123707,61729,-118495,-94770,0
C00682=28934,51901,-123680,61751,-118501,-94760,0
C00683=28915,51910,-123648,61776,-118507,-94748,0
C00684=28896,51919,-123617,61801,-118514,-94737,0
C00685=28877,51928,-123585,61826,-118520,-94725,0
C00686=28859,51937,-123553,61851,-118527,-94713,0
C00687=28840,51946,-123520,61876,-118533,-94702,0
C00688=28819,51956,-123483,61904,-118542,-94688,0
C00689=28798,51967,-123443,61931,-118551,-94675,0
C00690=28776,51980,-123399,61962,-118562,-94659,0
C00691=28752,51994,-123349,61995,-118573,-94641,0
C00692=28740,52000,-123329,62010,-118578,-94634,0
C00693=28717,52013,-123280,62042,-118589,-94617,0
C00694=28693,52026,-123233,62075,-118600,-94601,0
C00695=28672,52039,-123187,62103,-118611,-94585,0
C00696=28671,52044,-123169,62107,-118618,-94579,0
C00697=28669,52050,-123150,62111,-118625,-94574,0
C00698=28668,52055,-123132,62115,-118632,-94568,0
C00699=28666,52060,-123114,62119,-118639,-94563,0
C00700=28665,52065,-123095,62124,-118646,-94557,0
C00701=28663,52071,-123077,62128,-118653,-94552,0
C00702=28662,52076,-123057,62132,-118660,-94546,0
C00703=28660,52081,-123039,62136,-118666,-94541,0
C00704=28659,52086,-123021,62140,-118673,-94535,0
C00705=28657,52092,-123002,62144,-118680,-94530,0
C00706=28656,52097,-122983,62148,-118687,-94524,0
C00707=28655,52103,-122963,62152,-118695,-94518,0
C00708=28654,52108,-122944,62155,-118703,-94513,0
C00709=28653,52114,-122923,62159,-118710,-94507,0
C00710=28652,52120,-122903,62163,-118718,-94501,0
C00711=28651,52126,-122882,62166,-118726,-94495,0
C00712=28651,52132,-122860,62169,-118735,-94488,0
C00713=28650,52138,-122838,62173,-118743,-94482,0
C00714=28650,52145,-122816,62176,-118753,-94476,0
C00715=28650,52151,-122794,62179,-118761,-94469,0
C00716=28649,52157,-122771,62183,-118770,-94463,0
C00717=28649,52164,-122749,62186,-118778,-94456,0
C00718=28648,52170,-122728,62189,-118787,-94450,0
C00719=28648,52176,-122706,62193,-118796,-94444,0
C00720=28648,52183,-122683,62196,-118804,-94437,0
C00721=28647,52189,-122661,62199,-118813,-94431,0
C00722=28647,52195,-122639,62203,-118822,-94425,0
C00723=28651,52271,-122376,62233,-118927,-94350,0
C00724=28654,52346,-122113,62264,-119033,-94276,0
C00725=28656,52384,-121982,62279,-119086,-94238,0
C00726=22563,60493,-97223,72608,-124356,-86302,0
C00727=22464,60554,-97053,72736,-124343,-86238,0
C00728=22366,60614,-96883,72865,-124329,-86174,0
C00729=22267,60676,-96712,72994,-124317,-86110,0
C00730=22258,60682,-96695,73005,-124316,-86103,0
C00731=22250,60688,-96678,73017,-124316,-86097,0
C00732=22241,60694,-96661,73029,-124314,-86091,0
C00733=22232,60700,-96644,73041,-124313,-86085,0
C00734=22223,60706,-96627,73053,-124313,-86078,0
C00735=22214,60712,-96610,73064,-124312,-86072,0
C00736=22206,60718,-96593,73076,-124311,-86066,0
C00737=22197,60724,-96576,73088,-124311,-86060,0
C00738=22188,60731,-96559,73100,-124310,-86054,0
C00739=22180,60737,-96542,73111,-124310,-86048,0
C00740=22175,60740,-96534,73117,-124309,-86044,0
C00741=22157,60785,-96407,73157,-124332,-86005,0
C00742=22145,60821,-96307,73186,-124351,-85976,0
C00743=22137,60850,-96227,73208,-124367,-85951,0
C00744=22129,60879,-96146,73231,-124383,-85927,0
C00745=22122,60909,-96065,73252,-124401,-85903,0
C00746=22114,60938,-95984,73275,-124417,-85879,0
C00747=22109,60959,-95926,73289,-124429,-85861,0
C00748=22105,60980,-95867,73304,-124442,-85844,0
C00749=22102,60999,-95815,73316,-124454,-85829,0
C00750=22099,61018,-95763,73328,-124466,-85814,0
C00751=22096,61036,-95712,73340,-124478,-85799,0
C00752=22094,61055,-95660,73352,-124489,-85784,0
C00753=22091,61074,-95608,73364,-124502,-85769,0
C00754=22088,61093,-95556,73376,-124513,-85754,0
C00755=22086,61110,-95509,73386,-124525,-85740,0
C00756=22085,61125,-95468,73395,-124534,-85728,0
C00757=22083,61140,-95426,73404,-124544,-85716,0
C00758=22082,61155,-95385,73412,-124555,-85704,0
C00759=22081,61169,-95345,73420,-124564,-85693,0
C00760=22081,61183,-95306,73427,-124574,-85682,0
C00761=22080,61198,-95268,73435,-124583,-85671,0
C00762=22080,61212,-95228,73442,-124594,-85660,0
C00763=22079,61226,-95190,73449,-124604,-85649,0
C00764=22079,61240,-95151,73457,-124613,-85637,0
C00765=22078,61254,-95111,73464,-124624,-85626,0
C00766=22078,61268,-95072,73472,-124633,-85615,0
C00767=22077,61283,-95033,73479,-124643,-85604,0
C00768=22077,61296,-94997,73486,-124652,-85593,0
C00769=22077,61316,-94943,73496,-124666,-85578,0
C00770=22088,61325,-94917,73489,-124680,-85573,0
C00771=22099,61334,-94892,73482,-124694,-85567,0
C00772=22111,61343,-94867,73475,-124706,-85562,0
C00773=22122,61353,-94841,73468,-124721,-85557,0
C00774=22134,61362,-94815,73461,-124735,-85552,0
C00775=22146,61372,-94790,73454,-124749,-85546,0
C00776=22158,61381,-94764,73447,-124763,-85541,0
C00777=22170,61390,-94738,73440,-124776,-85535,0
C00778=22181,61399,-94714,73432,-124790,-85531,0
C00779=22193,61408,-94691,73426,-124803,-85526,0
C00780=22204,61416,-94668,73419,-124816,-85521,0
C00781=22219,61427,-94639,73409,-124832,-85515,0
C00782=22234,61437,-94610,73399,-124849,-85510,0
C00783=22251,61449,-94579,73388,-124867,-85503,0
C00784=22269,61461,-94547,73375,-124888,-85497,0
C00785=22288,61473,-94513,73363,-124907,-85491,0
C00786=22311,61486,-94477,73347,-124930,-85484,0
C00787=22334,61499,-94441,73330,-124955,-85478,0
C00788=22356,61513,-94405,73314,-124978,-85472,0
C00789=22379,61526,-94369,73298,-125002,-85465,0
C00790=22402,61539,-94332,73282,-125025,-85459,0
C00791=22431,61554,-94292,73261,-125053,-85452,0
C00792=22468,61573,-94241,73233,-125089,-85444,0
C00793=22515,61595,-94182,73198,-125134,-85435,0
C00794=22561,61616,-94123,73162,-125178,-85426,0
C00795=22579,61625,-94101,73148,-125195,-85422,0
C00796=22584,61624,-94102,73143,-125197,-85423,0
C00797=22594,61623,-94105,73133,-125203,-85426,0
C00798=22604,61622,-94107,73123,-125207,-85429,0
C00799=22614,61621,-94110,73112,-125213,-85431,0
C00800=22625,61620,-94114,73100,-125219,-85434,0
C00801=22636,61619,-94118,73089,-125225,-85437,0
C00802=22647,61617,-94121,73077,-125232,-85440,0
C00803=22658,61616,-94125,73065,-125237,-85443,0
C00804=22669,61615,-94129,73054,-125243,-85445,0
C00805=22680,61613,-94133,73042,-125249,-85448,0
C00806=22692,61612,-94136,73031,-125255,-85451,0
C00807=22703,61611,-94140,73019,-125260,-85454,0
C00808=22714,61610,-94143,73007,-125266,-85456,0
C00809=22725,61608,-94147,72996,-125272,-85459,0
C00810=22736,61607,-94151,72984,-125277,-85462,0
C00811=22747,61606,-94154,72973,-125283,-85465,0
C00812=22819,61595,-94186,72895,-125320,-85486,0
C00813=22952,61574,-94245,72752,-125386,-85525,0
C00814=23085,61553,-94303,72609,-125451,-85564,0
C00815=38484,60676,-96964,77281,-121845,-85584,0
C00816=38526,60774,-96692,77283,-121933,-85511,0
C00817=38568,60873,-96419,77285,-122022,-85438,0
C00818=38610,60972,-96145,77287,-122112,-85365,0
C00819=38615,60981,-96121,77287,-122120,-85358,0
C00820=38619,60990,-96095,77287,-122128,-85352,0
C00821=38623,60999,-96070,77286,-122137,-85345,0
C00822=38628,61008,-96045,77286,-122145,-85339,0
C00823=38632,61017,-96020,77286,-122154,-85332,0
C00824=38637,61027,-95995,77286,-122162,-85325,0
C00825=38641,61036,-95970,77285,-122170,-85319,0
C00826=38646,61045,-95945,77285,-122179,-85312,0
C00827=38650,61054,-95920,77285,-122187,-85306,0
C00828=38654,61063,-95896,77284,-122195,-85299,0
C00829=38657,61067,-95883,77284,-122200,-85296,0
C00830=38702,61096,-95806,77252,-122246,-85280,0
C00831=38739,61116,-95750,77225,-122282,-85269,0
C00832=38769,61131,-95709,77203,-122309,-85261,0
C00833=38799,61146,-95668,77180,-122338,-85254,0
C00834=38828,61161,-95627,77158,-122366,-85246,0
C00835=38858,61176,-95586,77135,-122393,-85239,0
C00836=38880,61186,-95559,77118,-122414,-85234,0
C00837=38902,61196,-95532,77101,-122433,-85230,0
C00838=38922,61204,-95510,77085,-122451,-85226,0
C00839=38942,61212,-95489,77070,-122468,-85223,0
C00840=38961,61220,-95468,77054,-122485,-85220,0
C00841=38981,61228,-95447,77038,-122502,-85216,0
C00842=39001,61236,-95425,77022,-122518,-85213,0
C00843=39020,61243,-95404,77007,-122536,-85210,0
C00844=39038,61250,-95385,76992,-122552,-85207,0
C00845=39054,61256,-95370,76979,-122565,-85205,0
C00846=39070,61262,-95355,76966,-122578,-85203,0
C00847=39086,61267,-95340,76953,-122592,-85201,0
C00848=39102,61272,-95327,76940,-122605,-85199,0
C00849=39117,61276,-95315,76927,-122616,-85198,0
C00850=39132,61281,-95302,76914,-122629,-85196,0
C00851=39147,61286,-95290,76902,-122641,-85195,0
C00852=39162,61290,-95278,76889,-122653,-85194,0
C00853=39177,61295,-95265,76876,-122665,-85192,0
C00854=39193,61300,-95253,76863,-122678,-85191,0
C00855=39208,61304,-95240,76851,-122691,-85190,0
C00856=39223,61309,-95228,76838,-122702,-85188,0
C00857=39237,61313,-95217,76826,-122714,-85187,0
C00858=39258,61319,-95201,76808,-122731,-85185,0
C00859=39271,61312,-95220,76792,-122734,-85193,0
C00860=39285,61305,-95238,76776,-122739,-85200,0
C00861=39298,61298,-95258,76760,-122742,-85208,0
C00862=39311,61291,-95279,76743,-122746,-85216,0
C00863=39325,61284,-95299,76727,-122749,-85223,0
C00864=39338,61276,-95319,76710,-122753,-85231,0
C00865=39352,61269,-95339,76694,-122756,-85239,0
C00866=39365,61262,-95360,76677,-122760,-85247,0
C00867=39378,61255,-95380,76662,-122763,-85255,0
C00868=39390,61248,-95399,76647,-122767,-85261,0
C00869=39402,61241,-95419,76631,-122769,-85269,0
C00870=39418,61231,-95446,76612,-122772,-85279,0
C00871=39434,61222,-95472,76592,-122776,-85289,0
C00872=39451,61211,-95503,76570,-122779,-85300,0
C00873=39469,61198,-95537,76547,-122783,-85313,0
C00874=39487,61186,-95572,76523,-122786,-85325,0
C00875=39508,61170,-95615,76496,-122788,-85341,0
C00876=39529,61155,-95658,76468,-122791,-85356,0
C00877=39549,61140,-95701,76441,-122794,-85372,0
C00878=39570,61124,-95744,76413,-122796,-85387,0
C00879=39591,61109,-95787,76386,-122799,-85402,0
C00880=39615,61089,-95842,76353,-122801,-85422,0
C00881=39646,61063,-95915,76311,-122802,-85447,0
C00882=39682,61030,-96007,76260,-122803,-85479,0
C00883=39719,60997,-96098,76209,-122803,-85510,0
C00884=39733,60984,-96135,76189,-122803,-85523,0
C00885=39734,60980,-96147,76186,-122801,-85527,0
C00886=39736,60971,-96169,76181,-122796,-85533,0
C00887=39738,60963,-96192,76175,-122793,-85540,0
C00888=39739,60954,-96217,76169,-122788,-85548,0
C00889=39741,60944,-96244,76163,-122783,-85556,0
C00890=39743,60935,-96271,76157,-122777,-85563,0
C00891=39745,60925,-96298,76151,-122772,-85571,0
C00892=39747,60915,-96325,76144,-122767,-85579,0
C00893=39748,60906,-96352,76138,-122761,-85588,0
C00894=39750,60896,-96378,76132,-122756,-85595,0
C00895=39752,60886,-96405,76126,-122750,-85603,0
C00896=39754,60876,-96432,76120,-122745,-85611,0
C00897=39756,60867,-96459,76113,-122740,-85620,0
C00898=39757,60857,-96486,76107,-122734,-85628,0
C00899=39759,60847,-96513,76101,-122729,-85635,0
C00900=39761,60838,-96540,76095,-122724,-85643,0
C00901=39769,60774,-96716,76058,-122686,-85696,0
C00902=39785,60657,-97042,75989,-122617,-85791,0
C00903=39800,60540,-97366,75921,-122548,-85886,0
C00904=37388,58322,-103607,77372,-119655,-87372,0
C00905=42893,55691,-111552,70547,-120342,-90429,0
C00906=44082,55209,-113072,69064,-120412,-91035,0
C00907=26167,57467,-105904,67398,-123765,-89337,0
C00908=27033,56739,-108074,66119,-123477,-90086,0
C00909=31664,53876,-117043,59673,-122149,-93308,0
C00910=30428,53970,-116713,61080,-121809,-93023,0
C00911=38802,58260,-103812,75918,-120391,-87615,0
C00912=39431,58256,-103839,75277,-120731,-87707,0
C00913=39809,58310,-103689,74917,-120976,-87715,0
C00914=45624,54217,-116252,66953,-120024,-92170,0
C00915=45544,54119,-116565,66994,-119883,-92250,0
C00916=45432,53853,-117426,66993,-119541,-92484,0
C00917=45369,53560,-118388,66929,-119184,-92756,0
C00918=45435,53180,-119655,66686,-118765,-93135,0
C00919=45591,52922,-120527,66400,-118516,-93410,0
C00920=31809,54181,-116059,59663,-122601,-93065,0
C00921=31653,54245,-115851,59866,-122624,-92984,0
C00922=31199,54365,-115457,60426,-122603,-92803,0
C00923=30676,54470,-115113,61053,-122531,-92624,0
C00924=30676,54411,-115136,61063,-122557,-92606,0
C00925=46667,54009,-116781,65762,-120296,-92442,0
C00926=46449,53707,-117756,65859,-119864,-92692,0
C00927=46352,53413,-118719,65830,-119482,-92956,0
C00928=46371,53124,-119683,65678,-119143,-93238,0
C00929=46505,52850,-120608,65407,-118858,-93525,0
C00930=46767,52586,-121515,65000,-118620,-93823,0
C00931=31615,53317,-118696,59495,-121497,-93725,0
C00932=31115,53498,-118093,60135,-121558,-93483,0
C00933=30590,53620,-117683,60772,-121525,-93289,0
C00934=30035,53688,-117451,61415,-121406,-93140,0
C00935=29469,53700,-117401,62042,-121207,-93041,0
C00936=28874,53653,-117543,62671,-120923,-92991,0
C00937=24551,59385,-100227,70075,-124678,-87453,0
C00938=24900,59663,-99448,69855,-125102,-87294,0
C00939=25167,59990,-98532,69747,-125521,-87083,0
C00940=25348,60363,-97493,69752,-125929,-86825,0
C00941=25435,60768,-96372,69872,-126306,-86528,0
C00942=29616,55183,-112694,84138,-113618,-89297,0
C00943=37714,58789,-102135,77270,-120206,-86957,0
C00944=38134,58587,-102721,76764,-120306,-87183,0
C00945=38596,58459,-103099,76244,-120474,-87354,0
C00946=39089,58405,-103263,75723,-120708,-87468,0
C00947=39591,58430,-103203,75224,-121003,-87519,0
C00948=40109,58539,-102901,74747,-121367,-87503,0
C00949=46596,54045,-116660,65857,-120310,-92397,0
C00950=48086,52592,-121532,63555,-119084,-94000,0
C00951=31387,52710,-120727,59456,-120581,-94246,0
C00952=31236,52828,-120325,59680,-120694,-94113,0
C00953=30961,52971,-119836,60052,-120796,-93938,0
C00954=30637,53086,-119446,60464,-120838,-93782,0
C00955=30278,53168,-119166,60899,-120820,-93652,0
C00956=29897,53213,-119009,61340,-120742,-93551,0
C00957=29509,53221,-118976,61770,-120611,-93485,0
C00958=29127,53192,-119065,62176,-120434,-93454,0
C00959=28765,53127,-119274,62542,-120219,-93461,0
C00960=28460,53037,-119570,62835,-119991,-93501,0
C00961=23543,59645,-99479,71237,-124326,-87075,0
C00962=23749,59738,-99221,71072,-124516,-87036,0
C00963=23797,59753,-99180,71031,-124555,-87032,0
C00964=24065,59893,-98791,70826,-124818,-86968,0
C00965=24295,60077,-98279,70684,-125096,-86862,0
C00966=24475,60298,-97663,70612,-125375,-86721,0
C00967=24600,60550,-96964,70612,-125648,-86546,0
C00968=24663,60824,-96207,70688,-125899,-86345,0
C00969=24662,61107,-95427,70835,-126119,-86127,0
C00970=24596,61389,-94649,71047,-126298,-85898,0
C00971=24504,61585,-94111,71241,-126391,-85731,0
C00972=37803,59627,-99759,77534,-120811,-86276,0
C00973=37962,59489,-100152,77317,-120814,-86412,0
C00974=37991,59455,-100247,77274,-120808,-86443,0
C00975=38222,59280,-100747,76969,-120826,-86619,0
C00976=38496,59146,-101132,76638,-120893,-86768,0
C00977=38802,59060,-101385,76294,-121008,-86883,0
C00978=39130,59023,-101496,75949,-121169,-86960,0
C00979=39464,59039,-101455,75620,-121369,-86994,0
C00980=39789,59109,-101263,75324,-121602,-86984,0
C00981=40091,59230,-100926,75073,-121860,-86930,0
C00982=40287,59353,-100582,74931,-122059,-86858,0
C00983=47881,54076,-116594,64473,-120850,-92563,0
C00984=47692,53964,-116952,64626,-120645,-92637,0
C00985=47486,53785,-117530,64766,-120353,-92772,0
C00986=47351,53591,-118158,64824,-120072,-92933,0
C00987=47291,53393,-118812,64797,-119810,-93111,0
C00988=47310,53197,-119464,64686,-119578,-93301,0
C00989=47406,53012,-120087,64495,-119383,-93493,0
C00990=47576,52844,-120658,64232,-119232,-93681,0
C00991=47813,52700,-121157,63905,-119130,-93856,0
C00992=48007,52623,-121424,63656,-119097,-93959,0
C00993=48200,53164,-119601,63694,-119859,-93463,0
C00994=48298,53068,-119922,63542,-119774,-93568,0
C00995=48432,52987,-120202,63357,-119717,-93666,0
C00996=48595,52922,-120425,63148,-119690,-93753,0
C00997=48695,52896,-120514,63026,-119693,-93791,0
C00998=48725,52886,-120551,62988,-119689,-93806,0
C00999=48913,52845,-120694,62763,-119701,-93873,0
C01000=49113,52823,-120774,62531,-119741,-93923,0
C01001=49650,52818,-120808,61937,-119918,-94008,0
C01002=30771,52081,-122883,59842,-119474,-94754,0
//INST
///DATE 2025/02/20 16:20
///COMM Generated using RoboDK
///ATTR SC,RW
///GROUP1 RB1
NOP
MOVL C00000 V=30.0 PL=1
MOVL C00001 V=30.0 PL=1
MOVL C00002 V=30.0 PL=1
MOVL C00003 V=30.0 PL=1
MOVL C00004 V=30.0 PL=1
MOVL C00005 V=30.0 PL=1
MOVL C00006 V=30.0 PL=1
MOVL C00007 V=30.0 PL=1
MOVL C00008 V=30.0 PL=1
MOVL C00009 V=30.0 PL=1
MOVL C00010 V=30.0 PL=1
MOVL C00011 V=30.0 PL=1
MOVL C00012 V=30.0 PL=1
MOVL C00013 V=30.0 PL=1
MOVL C00014 V=30.0 PL=1
MOVL C00015 V=30.0 PL=1
MOVL C00016 V=30.0 PL=1
MOVL C00017 V=30.0 PL=1
MOVL C00018 V=30.0 PL=1
MOVL C00019 V=30.0 PL=1
MOVL C00020 V=30.0 PL=1
MOVL C00021 V=30.0 PL=1
MOVL C00022 V=30.0 PL=1
MOVL C00023 V=30.0 PL=1
MOVL C00024 V=30.0 PL=1
MOVL C00025 V=30.0 PL=1
MOVL C00026 V=30.0 PL=1
MOVL C00027 V=30.0 PL=1
MOVL C00028 V=30.0 PL=1
MOVL C00029 V=30.0 PL=1
MOVL C00030 V=30.0 PL=1
MOVL C00031 V=30.0 PL=1
MOVL C00032 V=30.0 PL=1
MOVL C00033 V=30.0 PL=1
MOVL C00034 V=30.0 PL=1
MOVL C00035 V=30.0 PL=1
MOVL C00036 V=30.0 PL=1
MOVL C00037 V=30.0 PL=1
MOVL C00038 V=30.0 PL=1
MOVL C00039 V=30.0 PL=1
MOVL C00040 V=30.0 PL=1
MOVL C00041 V=30.0 PL=1
MOVL C00042 V=30.0 PL=1
MOVL C00043 V=30.0 PL=1
MOVL C00044 V=30.0 PL=1
MOVL C00045 V=30.0 PL=1
MOVL C00046 V=30.0 PL=1
MOVL C00047 V=30.0 PL=1
MOVL C00048 V=30.0 PL=1
MOVL C00049 V=30.0 PL=1
MOVL C00050 V=30.0 PL=1
MOVL C00051 V=30.0 PL=1
MOVL C00052 V=30.0 PL=1
MOVL C00053 V=30.0 PL=1
MOVL C00054 V=30.0 PL=1
MOVL C00055 V=30.0 PL=1
MOVL C00056 V=30.0 PL=1
MOVL C00057 V=30.0 PL=1
MOVL C00058 V=30.0 PL=1
MOVL C00059 V=30.0 PL=1
MOVL C00060 V=30.0 PL=1
MOVL C00061 V=30.0 PL=1
MOVL C00062 V=30.0 PL=1
MOVL C00063 V=30.0 PL=1
MOVL C00064 V=30.0 PL=1
MOVL C00065 V=30.0 PL=1
MOVL C00066 V=30.0 PL=1
MOVL C00067 V=30.0 PL=1
MOVL C00068 V=30.0 PL=1
MOVL C00069 V=30.0 PL=1
MOVL C00070 V=30.0 PL=1
MOVL C00071 V=30.0 PL=1
MOVL C00072 V=30.0 PL=1
MOVL C00073 V=30.0 PL=1
MOVL C00074 V=30.0 PL=1
MOVL C00075 V=30.0 PL=1
MOVL C00076 V=30.0 PL=1
MOVL C00077 V=30.0 PL=1
MOVL C00078 V=30.0 PL=1
MOVL C00079 V=30.0 PL=1
MOVL C00080 V=30.0 PL=1
MOVL C00081 V=30.0 PL=1
MOVL C00082 V=30.0 PL=1
MOVL C00083 V=30.0 PL=1
MOVL C00084 V=30.0 PL=1
MOVL C00085 V=30.0 PL=1
MOVL C00086 V=30.0 PL=1
MOVL C00087 V=30.0 PL=1
MOVL C00088 V=30.0 PL=1
MOVL C00089 V=30.0 PL=1
MOVL C00090 V=30.0 PL=1
MOVL C00091 V=30.0 PL=1
MOVL C00092 V=30.0 PL=1
MOVL C00093 V=30.0 PL=1
MOVL C00094 V=30.0 PL=1
MOVL C00095 V=30.0 PL=1
MOVL C00096 V=30.0 PL=1
MOVL C00097 V=30.0 PL=1
MOVL C00098 V=30.0 PL=1
MOVL C00099 V=30.0 PL=1
MOVL C00100 V=30.0 PL=1
MOVL C00101 V=30.0 PL=1
MOVL C00102 V=30.0 PL=1
MOVL C00103 V=30.0 PL=1
MOVL C00104 V=30.0 PL=1
MOVL C00105 V=30.0 PL=1
MOVL C00106 V=30.0 PL=1
MOVL C00107 V=130.0 PL=1
MOVL C00108 V=30.0 PL=1
MOVL C00109 V=30.0 PL=1
MOVL C00110 V=30.0 PL=1
MOVL C00111 V=30.0 PL=1
MOVL C00112 V=30.0 PL=1
MOVL C00113 V=30.0 PL=1
MOVL C00114 V=30.0 PL=1
MOVL C00115 V=30.0 PL=1
MOVL C00116 V=30.0 PL=1
MOVL C00117 V=30.0 PL=1
MOVL C00118 V=30.0 PL=1
MOVL C00119 V=30.0 PL=1
MOVL C00120 V=30.0 PL=1
MOVL C00121 V=30.0 PL=1
MOVL C00122 V=30.0 PL=1
MOVL C00123 V=30.0 PL=1
MOVL C00124 V=30.0 PL=1
MOVL C00125 V=30.0 PL=1
MOVL C00126 V=30.0 PL=1
MOVL C00127 V=30.0 PL=1
MOVL C00128 V=30.0 PL=1
MOVL C00129 V=30.0 PL=1
MOVL C00130 V=30.0 PL=1
MOVL C00131 V=30.0 PL=1
MOVL C00132 V=30.0 PL=1
MOVL C00133 V=30.0 PL=1
MOVL C00134 V=30.0 PL=1
MOVL C00135 V=30.0 PL=1
MOVL C00136 V=30.0 PL=1
MOVL C00137 V=30.0 PL=1
MOVL C00138 V=30.0 PL=1
MOVL C00139 V=30.0 PL=1
MOVL C00140 V=30.0 PL=1
MOVL C00141 V=30.0 PL=1
MOVL C00142 V=30.0 PL=1
MOVL C00143 V=30.0 PL=1
MOVL C00144 V=30.0 PL=1
MOVL C00145 V=30.0 PL=1
MOVL C00146 V=30.0 PL=1
MOVL C00147 V=30.0 PL=1
MOVL C00148 V=30.0 PL=1
MOVL C00149 V=30.0 PL=1
MOVL C00150 V=30.0 PL=1
MOVL C00151 V=30.0 PL=1
MOVL C00152 V=30.0 PL=1
MOVL C00153 V=30.0 PL=1
MOVL C00154 V=30.0 PL=1
MOVL C00155 V=30.0 PL=1
MOVL C00156 V=30.0 PL=1
MOVL C00157 V=30.0 PL=1
MOVL C00158 V=30.0 PL=1
MOVL C00159 V=30.0 PL=1
MOVL C00160 V=30.0 PL=1
MOVL C00161 V=30.0 PL=1
MOVL C00162 V=30.0 PL=1
MOVL C00163 V=30.0 PL=1
MOVL C00164 V=30.0 PL=1
MOVL C00165 V=30.0 PL=1
MOVL C00166 V=30.0 PL=1
MOVL C00167 V=30.0 PL=1
MOVL C00168 V=30.0 PL=1
MOVL C00169 V=30.0 PL=1
MOVL C00170 V=30.0 PL=1
MOVL C00171 V=30.0 PL=1
MOVL C00172 V=30.0 PL=1
MOVL C00173 V=30.0 PL=1
MOVL C00174 V=30.0 PL=1
MOVL C00175 V=30.0 PL=1
MOVL C00176 V=30.0 PL=1
MOVL C00177 V=30.0 PL=1
MOVL C00178 V=30.0 PL=1
MOVL C00179 V=30.0 PL=1
MOVL C00180 V=30.0 PL=1
MOVL C00181 V=30.0 PL=1
MOVL C00182 V=30.0 PL=1
MOVL C00183 V=30.0 PL=1
MOVL C00184 V=30.0 PL=1
MOVL C00185 V=30.0 PL=1
MOVL C00186 V=30.0 PL=1
MOVL C00187 V=30.0 PL=1
MOVL C00188 V=30.0 PL=1
MOVL C00189 V=30.0 PL=1
MOVL C00190 V=30.0 PL=1
MOVL C00191 V=30.0 PL=1
MOVL C00192 V=30.0 PL=1
MOVL C00193 V=30.0 PL=1
MOVL C00194 V=30.0 PL=1
MOVL C00195 V=30.0 PL=1
MOVL C00196 V=30.0 PL=1
MOVL C00197 V=30.0 PL=1
MOVL C00198 V=130.0 PL=1
MOVL C00199 V=30.0 PL=1
MOVL C00200 V=30.0 PL=1
MOVL C00201 V=30.0 PL=1
MOVL C00202 V=30.0 PL=1
MOVL C00203 V=30.0 PL=1
MOVL C00204 V=30.0 PL=1
MOVL C00205 V=30.0 PL=1
MOVL C00206 V=30.0 PL=1
MOVL C00207 V=30.0 PL=1
MOVL C00208 V=30.0 PL=1
MOVL C00209 V=30.0 PL=1
MOVL C00210 V=30.0 PL=1
MOVL C00211 V=30.0 PL=1
MOVL C00212 V=30.0 PL=1
MOVL C00213 V=30.0 PL=1
MOVL C00214 V=30.0 PL=1
MOVL C00215 V=30.0 PL=1
MOVL C00216 V=30.0 PL=1
MOVL C00217 V=30.0 PL=1
MOVL C00218 V=30.0 PL=1
MOVL C00219 V=30.0 PL=1
MOVL C00220 V=30.0 PL=1
MOVL C00221 V=30.0 PL=1
MOVL C00222 V=30.0 PL=1
MOVL C00223 V=30.0 PL=1
MOVL C00224 V=30.0 PL=1
MOVL C00225 V=30.0 PL=1
MOVL C00226 V=30.0 PL=1
MOVL C00227 V=30.0 PL=1
MOVL C00228 V=30.0 PL=1
MOVL C00229 V=30.0 PL=1
MOVL C00230 V=30.0 PL=1
MOVL C00231 V=30.0 PL=1
MOVL C00232 V=30.0 PL=1
MOVL C00233 V=30.0 PL=1
MOVL C00234 V=30.0 PL=1
MOVL C00235 V=30.0 PL=1
MOVL C00236 V=30.0 PL=1
MOVL C00237 V=30.0 PL=1
MOVL C00238 V=30.0 PL=1
MOVL C00239 V=30.0 PL=1
MOVL C00240 V=30.0 PL=1
MOVL C00241 V=30.0 PL=1
MOVL C00242 V=30.0 PL=1
MOVL C00243 V=30.0 PL=1
MOVL C00244 V=30.0 PL=1
MOVL C00245 V=30.0 PL=1
MOVL C00246 V=30.0 PL=1
MOVL C00247 V=30.0 PL=1
MOVL C00248 V=30.0 PL=1
MOVL C00249 V=30.0 PL=1
MOVL C00250 V=30.0 PL=1
MOVL C00251 V=30.0 PL=1
MOVL C00252 V=30.0 PL=1
MOVL C00253 V=30.0 PL=1
MOVL C00254 V=30.0 PL=1
MOVL C00255 V=30.0 PL=1
MOVL C00256 V=30.0 PL=1
MOVL C00257 V=30.0 PL=1
MOVL C00258 V=30.0 PL=1
MOVL C00259 V=30.0 PL=1
MOVL C00260 V=30.0 PL=1
MOVL C00261 V=30.0 PL=1
MOVL C00262 V=30.0 PL=1
MOVL C00263 V=30.0 PL=1
MOVL C00264 V=30.0 PL=1
MOVL C00265 V=30.0 PL=1
MOVL C00266 V=30.0 PL=1
MOVL C00267 V=30.0 PL=1
MOVL C00268 V=30.0 PL=1
MOVL C00269 V=30.0 PL=1
MOVL C00270 V=30.0 PL=1
MOVL C00271 V=30.0 PL=1
MOVL C00272 V=30.0 PL=1
MOVL C00273 V=30.0 PL=1
MOVL C00274 V=30.0 PL=1
MOVL C00275 V=30.0 PL=1
MOVL C00276 V=30.0 PL=1
MOVL C00277 V=30.0 PL=1
MOVL C00278 V=30.0 PL=1
MOVL C00279 V=30.0 PL=1
MOVL C00280 V=30.0 PL=1
MOVL C00281 V=30.0 PL=1
MOVL C00282 V=30.0 PL=1
MOVL C00283 V=30.0 PL=1
MOVL C00284 V=30.0 PL=1
MOVL C00285 V=30.0 PL=1
MOVL C00286 V=30.0 PL=1
MOVL C00287 V=30.0 PL=1
MOVL C00288 V=30.0 PL=1
MOVL C00289 V=30.0 PL=1
MOVL C00290 V=30.0 PL=1
MOVL C00291 V=130.0 PL=1
MOVL C00292 V=20.0 PL=1
MOVL C00293 V=20.0 PL=1
MOVL C00294 V=20.0 PL=1
MOVL C00295 V=20.0 PL=1
MOVL C00296 V=20.0 PL=1
MOVL C00297 V=20.0 PL=1
MOVL C00298 V=20.0 PL=1
MOVL C00299 V=20.0 PL=1
MOVL C00300 V=20.0 PL=1
MOVL C00301 V=20.0 PL=1
MOVL C00302 V=20.0 PL=1
MOVL C00303 V=20.0 PL=1
MOVL C00304 V=20.0 PL=1
MOVL C00305 V=20.0 PL=1
MOVL C00306 V=20.0 PL=1
MOVL C00307 V=20.0 PL=1
MOVL C00308 V=20.0 PL=1
MOVL C00309 V=20.0 PL=1
MOVL C00310 V=20.0 PL=1
MOVL C00311 V=20.0 PL=1
MOVL C00312 V=20.0 PL=1
MOVL C00313 V=20.0 PL=1
MOVL C00314 V=20.0 PL=1
MOVL C00315 V=20.0 PL=1
MOVL C00316 V=20.0 PL=1
MOVL C00317 V=20.0 PL=1
MOVL C00318 V=20.0 PL=1
MOVL C00319 V=20.0 PL=1
MOVL C00320 V=20.0 PL=1
MOVL C00321 V=20.0 PL=1
MOVL C00322 V=20.0 PL=1
MOVL C00323 V=20.0 PL=1
MOVL C00324 V=20.0 PL=1
MOVL C00325 V=20.0 PL=1
MOVL C00326 V=20.0 PL=1
MOVL C00327 V=20.0 PL=1
MOVL C00328 V=20.0 PL=1
MOVL C00329 V=20.0 PL=1
MOVL C00330 V=20.0 PL=1
MOVL C00331 V=20.0 PL=1
MOVL C00332 V=20.0 PL=1
MOVL C00333 V=20.0 PL=1
MOVL C00334 V=20.0 PL=1
MOVL C00335 V=20.0 PL=1
MOVL C00336 V=130.0 PL=1
MOVL C00337 V=130.0 PL=1
MOVL C00338 V=60.0 PL=1
MOVL C00339 V=60.0 PL=1
MOVL C00340 V=60.0 PL=1
MOVL C00341 V=60.0 PL=1
MOVL C00342 V=60.0 PL=1
MOVL C00343 V=60.0 PL=1
MOVL C00344 V=60.0 PL=1
MOVL C00345 V=60.0 PL=1
MOVL C00346 V=60.0 PL=1
MOVL C00347 V=60.0 PL=1
MOVL C00348 V=60.0 PL=1
MOVL C00349 V=60.0 PL=1
MOVL C00350 V=60.0 PL=1
MOVL C00351 V=60.0 PL=1
MOVL C00352 V=60.0 PL=1
MOVL C00353 V=60.0 PL=1
MOVL C00354 V=60.0 PL=1
MOVL C00355 V=60.0 PL=1
MOVL C00356 V=60.0 PL=1
MOVL C00357 V=60.0 PL=1
MOVL C00358 V=60.0 PL=1
MOVL C00359 V=60.0 PL=1
MOVL C00360 V=60.0 PL=1
MOVL C00361 V=60.0 PL=1
MOVL C00362 V=60.0 PL=1
MOVL C00363 V=60.0 PL=1
MOVL C00364 V=60.0 PL=1
MOVL C00365 V=60.0 PL=1
MOVL C00366 V=130.0 PL=1
MOVL C00367 V=60.0 PL=1
MOVL C00368 V=60.0 PL=1
MOVL C00369 V=60.0 PL=1
MOVL C00370 V=60.0 PL=1
MOVL C00371 V=60.0 PL=1
MOVL C00372 V=60.0 PL=1
MOVL C00373 V=60.0 PL=1
MOVL C00374 V=60.0 PL=1
MOVL C00375 V=60.0 PL=1
MOVL C00376 V=60.0 PL=1
MOVL C00377 V=60.0 PL=1
MOVL C00378 V=60.0 PL=1
MOVL C00379 V=60.0 PL=1
MOVL C00380 V=60.0 PL=1
MOVL C00381 V=60.0 PL=1
MOVL C00382 V=60.0 PL=1
MOVL C00383 V=60.0 PL=1
MOVL C00384 V=60.0 PL=1
MOVL C00385 V=60.0 PL=1
MOVL C00386 V=60.0 PL=1
MOVL C00387 V=60.0 PL=1
MOVL C00388 V=60.0 PL=1
MOVL C00389 V=60.0 PL=1
MOVL C00390 V=60.0 PL=1
MOVL C00391 V=60.0 PL=1
MOVL C00392 V=60.0 PL=1
MOVL C00393 V=60.0 PL=1
MOVL C00394 V=60.0 PL=1
MOVL C00395 V=60.0 PL=1
MOVL C00396 V=60.0 PL=1
MOVL C00397 V=60.0 PL=1
MOVL C00398 V=60.0 PL=1
MOVL C00399 V=60.0 PL=1
MOVL C00400 V=60.0 PL=1
MOVL C00401 V=60.0 PL=1
MOVL C00402 V=60.0 PL=1
MOVL C00403 V=60.0 PL=1
MOVL C00404 V=60.0 PL=1
MOVL C00405 V=60.0 PL=1
MOVL C00406 V=60.0 PL=1
MOVL C00407 V=60.0 PL=1
MOVL C00408 V=60.0 PL=1
MOVL C00409 V=60.0 PL=1
MOVL C00410 V=60.0 PL=1
MOVL C00411 V=130.0 PL=1
MOVL C00412 V=30.0 PL=1
MOVL C00413 V=30.0 PL=1
MOVL C00414 V=30.0 PL=1
MOVL C00415 V=30.0 PL=1
MOVL C00416 V=30.0 PL=1
MOVL C00417 V=30.0 PL=1
MOVL C00418 V=30.0 PL=1
MOVL C00419 V=30.0 PL=1
MOVL C00420 V=30.0 PL=1
MOVL C00421 V=30.0 PL=1
MOVL C00422 V=30.0 PL=1
MOVL C00423 V=30.0 PL=1
MOVL C00424 V=30.0 PL=1
MOVL C00425 V=30.0 PL=1
MOVL C00426 V=30.0 PL=1
MOVL C00427 V=30.0 PL=1
MOVL C00428 V=30.0 PL=1
MOVL C00429 V=30.0 PL=1
MOVL C00430 V=30.0 PL=1
MOVL C00431 V=30.0 PL=1
MOVL C00432 V=30.0 PL=1
MOVL C00433 V=30.0 PL=1
MOVL C00434 V=30.0 PL=1
MOVL C00435 V=30.0 PL=1
MOVL C00436 V=30.0 PL=1
MOVL C00437 V=30.0 PL=1
MOVL C00438 V=30.0 PL=1
MOVL C00439 V=30.0 PL=1
MOVL C00440 V=30.0 PL=1
MOVL C00441 V=30.0 PL=1
MOVL C00442 V=30.0 PL=1
MOVL C00443 V=30.0 PL=1
MOVL C00444 V=30.0 PL=1
MOVL C00445 V=30.0 PL=1
MOVL C00446 V=30.0 PL=1
MOVL C00447 V=30.0 PL=1
MOVL C00448 V=30.0 PL=1
MOVL C00449 V=30.0 PL=1
MOVL C00450 V=30.0 PL=1
MOVL C00451 V=30.0 PL=1
MOVL C00452 V=30.0 PL=1
MOVL C00453 V=30.0 PL=1
MOVL C00454 V=30.0 PL=1
MOVL C00455 V=30.0 PL=1
MOVL C00456 V=30.0 PL=1
MOVL C00457 V=30.0 PL=1
MOVL C00458 V=30.0 PL=1
MOVL C00459 V=30.0 PL=1
MOVL C00460 V=30.0 PL=1
MOVL C00461 V=30.0 PL=1
MOVL C00462 V=30.0 PL=1
MOVL C00463 V=30.0 PL=1
MOVL C00464 V=30.0 PL=1
MOVL C00465 V=30.0 PL=1
MOVL C00466 V=30.0 PL=1
MOVL C00467 V=30.0 PL=1
MOVL C00468 V=30.0 PL=1
MOVL C00469 V=30.0 PL=1
MOVL C00470 V=30.0 PL=1
MOVL C00471 V=30.0 PL=1
MOVL C00472 V=30.0 PL=1
MOVL C00473 V=30.0 PL=1
MOVL C00474 V=30.0 PL=1
MOVL C00475 V=30.0 PL=1
MOVL C00476 V=30.0 PL=1
MOVL C00477 V=30.0 PL=1
MOVL C00478 V=30.0 PL=1
MOVL C00479 V=30.0 PL=1
MOVL C00480 V=30.0 PL=1
MOVL C00481 V=30.0 PL=1
MOVL C00482 V=30.0 PL=1
MOVL C00483 V=30.0 PL=1
MOVL C00484 V=130.0 PL=1
MOVL C00485 V=130.0 PL=1
MOVL C00486 V=30.0 PL=1
MOVL C00487 V=30.0 PL=1
MOVL C00488 V=30.0 PL=1
MOVL C00489 V=30.0 PL=1
MOVL C00490 V=30.0 PL=1
MOVL C00491 V=30.0 PL=1
MOVL C00492 V=30.0 PL=1
MOVL C00493 V=30.0 PL=1
MOVL C00494 V=30.0 PL=1
MOVL C00495 V=30.0 PL=1
MOVL C00496 V=30.0 PL=1
MOVL C00497 V=30.0 PL=1
MOVL C00498 V=30.0 PL=1
MOVL C00499 V=30.0 PL=1
MOVL C00500 V=30.0 PL=1
MOVL C00501 V=30.0 PL=1
MOVL C00502 V=30.0 PL=1
MOVL C00503 V=30.0 PL=1
MOVL C00504 V=30.0 PL=1
MOVL C00505 V=30.0 PL=1
MOVL C00506 V=30.0 PL=1
MOVL C00507 V=30.0 PL=1
MOVL C00508 V=30.0 PL=1
MOVL C00509 V=30.0 PL=1
MOVL C00510 V=30.0 PL=1
MOVL C00511 V=30.0 PL=1
MOVL C00512 V=30.0 PL=1
MOVL C00513 V=30.0 PL=1
MOVL C00514 V=30.0 PL=1
MOVL C00515 V=30.0 PL=1
MOVL C00516 V=30.0 PL=1
MOVL C00517 V=30.0 PL=1
MOVL C00518 V=30.0 PL=1
MOVL C00519 V=30.0 PL=1
MOVL C00520 V=30.0 PL=1
MOVL C00521 V=30.0 PL=1
MOVL C00522 V=30.0 PL=1
MOVL C00523 V=30.0 PL=1
MOVL C00524 V=30.0 PL=1
MOVL C00525 V=30.0 PL=1
MOVL C00526 V=30.0 PL=1
MOVL C00527 V=30.0 PL=1
MOVL C00528 V=30.0 PL=1
MOVL C00529 V=30.0 PL=1
MOVL C00530 V=30.0 PL=1
MOVL C00531 V=30.0 PL=1
MOVL C00532 V=30.0 PL=1
MOVL C00533 V=30.0 PL=1
MOVL C00534 V=30.0 PL=1
MOVL C00535 V=30.0 PL=1
MOVL C00536 V=30.0 PL=1
MOVL C00537 V=30.0 PL=1
MOVL C00538 V=30.0 PL=1
MOVL C00539 V=30.0 PL=1
MOVL C00540 V=30.0 PL=1
MOVL C00541 V=30.0 PL=1
MOVL C00542 V=30.0 PL=1
MOVL C00543 V=30.0 PL=1
MOVL C00544 V=30.0 PL=1
MOVL C00545 V=30.0 PL=1
MOVL C00546 V=30.0 PL=1
MOVL C00547 V=30.0 PL=1
MOVL C00548 V=30.0 PL=1
MOVL C00549 V=30.0 PL=1
MOVL C00550 V=30.0 PL=1
MOVL C00551 V=30.0 PL=1
MOVL C00552 V=30.0 PL=1
MOVL C00553 V=30.0 PL=1
MOVL C00554 V=30.0 PL=1
MOVL C00555 V=30.0 PL=1
MOVL C00556 V=30.0 PL=1
MOVL C00557 V=30.0 PL=1
MOVL C00558 V=30.0 PL=1
MOVL C00559 V=30.0 PL=1
MOVL C00560 V=30.0 PL=1
MOVL C00561 V=30.0 PL=1
MOVL C00562 V=30.0 PL=1
MOVL C00563 V=30.0 PL=1
MOVL C00564 V=30.0 PL=1
MOVL C00565 V=30.0 PL=1
MOVL C00566 V=30.0 PL=1
MOVL C00567 V=30.0 PL=1
MOVL C00568 V=30.0 PL=1
MOVL C00569 V=30.0 PL=1
MOVL C00570 V=30.0 PL=1
MOVL C00571 V=30.0 PL=1
MOVL C00572 V=30.0 PL=1
MOVL C00573 V=30.0 PL=1
MOVL C00574 V=30.0 PL=1
MOVL C00575 V=30.0 PL=1
MOVL C00576 V=30.0 PL=1
MOVL C00577 V=30.0 PL=1
MOVL C00578 V=30.0 PL=1
MOVL C00579 V=30.0 PL=1
MOVL C00580 V=30.0 PL=1
MOVL C00581 V=30.0 PL=1
MOVL C00582 V=30.0 PL=1
MOVL C00583 V=30.0 PL=1
MOVL C00584 V=30.0 PL=1
MOVL C00585 V=30.0 PL=1
MOVL C00586 V=30.0 PL=1
MOVL C00587 V=30.0 PL=1
MOVL C00588 V=30.0 PL=1
MOVL C00589 V=30.0 PL=1
MOVL C00590 V=30.0 PL=1
MOVL C00591 V=30.0 PL=1
MOVL C00592 V=30.0 PL=1
MOVL C00593 V=30.0 PL=1
MOVL C00594 V=30.0 PL=1
MOVL C00595 V=30.0 PL=1
MOVL C00596 V=30.0 PL=1
MOVL C00597 V=30.0 PL=1
MOVL C00598 V=30.0 PL=1
MOVL C00599 V=30.0 PL=1
MOVL C00600 V=30.0 PL=1
MOVL C00601 V=30.0 PL=1
MOVL C00602 V=30.0 PL=1
MOVL C00603 V=30.0 PL=1
MOVL C00604 V=30.0 PL=1
MOVL C00605 V=130.0 PL=1
MOVL C00606 V=30.0 PL=1
MOVL C00607 V=30.0 PL=1
MOVL C00608 V=30.0 PL=1
MOVL C00609 V=30.0 PL=1
MOVL C00610 V=30.0 PL=1
MOVL C00611 V=30.0 PL=1
MOVL C00612 V=30.0 PL=1
MOVL C00613 V=30.0 PL=1
MOVL C00614 V=30.0 PL=1
MOVL C00615 V=30.0 PL=1
MOVL C00616 V=30.0 PL=1
MOVL C00617 V=30.0 PL=1
MOVL C00618 V=30.0 PL=1
MOVL C00619 V=30.0 PL=1
MOVL C00620 V=30.0 PL=1
MOVL C00621 V=30.0 PL=1
MOVL C00622 V=30.0 PL=1
MOVL C00623 V=30.0 PL=1
MOVL C00624 V=30.0 PL=1
MOVL C00625 V=30.0 PL=1
MOVL C00626 V=30.0 PL=1
MOVL C00627 V=30.0 PL=1
MOVL C00628 V=30.0 PL=1
MOVL C00629 V=30.0 PL=1
MOVL C00630 V=30.0 PL=1
MOVL C00631 V=30.0 PL=1
MOVL C00632 V=30.0 PL=1
MOVL C00633 V=30.0 PL=1
MOVL C00634 V=30.0 PL=1
MOVL C00635 V=30.0 PL=1
MOVL C00636 V=30.0 PL=1
MOVL C00637 V=30.0 PL=1
MOVL C00638 V=30.0 PL=1
MOVL C00639 V=30.0 PL=1
MOVL C00640 V=30.0 PL=1
MOVL C00641 V=30.0 PL=1
MOVL C00642 V=30.0 PL=1
MOVL C00643 V=30.0 PL=1
MOVL C00644 V=30.0 PL=1
MOVL C00645 V=30.0 PL=1
MOVL C00646 V=30.0 PL=1
MOVL C00647 V=30.0 PL=1
MOVL C00648 V=30.0 PL=1
MOVL C00649 V=30.0 PL=1
MOVL C00650 V=30.0 PL=1
MOVL C00651 V=30.0 PL=1
MOVL C00652 V=30.0 PL=1
MOVL C00653 V=30.0 PL=1
MOVL C00654 V=30.0 PL=1
MOVL C00655 V=30.0 PL=1
MOVL C00656 V=30.0 PL=1
MOVL C00657 V=30.0 PL=1
MOVL C00658 V=30.0 PL=1
MOVL C00659 V=30.0 PL=1
MOVL C00660 V=30.0 PL=1
MOVL C00661 V=30.0 PL=1
MOVL C00662 V=30.0 PL=1
MOVL C00663 V=30.0 PL=1
MOVL C00664 V=30.0 PL=1
MOVL C00665 V=30.0 PL=1
MOVL C00666 V=30.0 PL=1
MOVL C00667 V=30.0 PL=1
MOVL C00668 V=30.0 PL=1
MOVL C00669 V=30.0 PL=1
MOVL C00670 V=30.0 PL=1
MOVL C00671 V=30.0 PL=1
MOVL C00672 V=30.0 PL=1
MOVL C00673 V=30.0 PL=1
MOVL C00674 V=30.0 PL=1
MOVL C00675 V=30.0 PL=1
MOVL C00676 V=30.0 PL=1
MOVL C00677 V=30.0 PL=1
MOVL C00678 V=30.0 PL=1
MOVL C00679 V=30.0 PL=1
MOVL C00680 V=30.0 PL=1
MOVL C00681 V=30.0 PL=1
MOVL C00682 V=30.0 PL=1
MOVL C00683 V=30.0 PL=1
MOVL C00684 V=30.0 PL=1
MOVL C00685 V=30.0 PL=1
MOVL C00686 V=30.0 PL=1
MOVL C00687 V=30.0 PL=1
MOVL C00688 V=30.0 PL=1
MOVL C00689 V=30.0 PL=1
MOVL C00690 V=30.0 PL=1
MOVL C00691 V=30.0 PL=1
MOVL C00692 V=30.0 PL=1
MOVL C00693 V=30.0 PL=1
MOVL C00694 V=30.0 PL=1
MOVL C00695 V=30.0 PL=1
MOVL C00696 V=30.0 PL=1
MOVL C00697 V=30.0 PL=1
MOVL C00698 V=30.0 PL=1
MOVL C00699 V=30.0 PL=1
MOVL C00700 V=30.0 PL=1
MOVL C00701 V=30.0 PL=1
MOVL C00702 V=30.0 PL=1
MOVL C00703 V=30.0 PL=1
MOVL C00704 V=30.0 PL=1
MOVL C00705 V=30.0 PL=1
MOVL C00706 V=30.0 PL=1
MOVL C00707 V=30.0 PL=1
MOVL C00708 V=30.0 PL=1
MOVL C00709 V=30.0 PL=1
MOVL C00710 V=30.0 PL=1
MOVL C00711 V=30.0 PL=1
MOVL C00712 V=30.0 PL=1
MOVL C00713 V=30.0 PL=1
MOVL C00714 V=30.0 PL=1
MOVL C00715 V=30.0 PL=1
MOVL C00716 V=30.0 PL=1
MOVL C00717 V=30.0 PL=1
MOVL C00718 V=30.0 PL=1
MOVL C00719 V=30.0 PL=1
MOVL C00720 V=30.0 PL=1
MOVL C00721 V=30.0 PL=1
MOVL C00722 V=30.0 PL=1
MOVL C00723 V=30.0 PL=1
MOVL C00724 V=30.0 PL=1
MOVL C00725 V=30.0 PL=1
MOVL C00726 V=130.0 PL=1
MOVL C00727 V=30.0 PL=1
MOVL C00728 V=30.0 PL=1
MOVL C00729 V=30.0 PL=1
MOVL C00730 V=30.0 PL=1
MOVL C00731 V=30.0 PL=1
MOVL C00732 V=30.0 PL=1
MOVL C00733 V=30.0 PL=1
MOVL C00734 V=30.0 PL=1
MOVL C00735 V=30.0 PL=1
MOVL C00736 V=30.0 PL=1
MOVL C00737 V=30.0 PL=1
MOVL C00738 V=30.0 PL=1
MOVL C00739 V=30.0 PL=1
MOVL C00740 V=30.0 PL=1
MOVL C00741 V=30.0 PL=1
MOVL C00742 V=30.0 PL=1
MOVL C00743 V=30.0 PL=1
MOVL C00744 V=30.0 PL=1
MOVL C00745 V=30.0 PL=1
MOVL C00746 V=30.0 PL=1
MOVL C00747 V=30.0 PL=1
MOVL C00748 V=30.0 PL=1
MOVL C00749 V=30.0 PL=1
MOVL C00750 V=30.0 PL=1
MOVL C00751 V=30.0 PL=1
MOVL C00752 V=30.0 PL=1
MOVL C00753 V=30.0 PL=1
MOVL C00754 V=30.0 PL=1
MOVL C00755 V=30.0 PL=1
MOVL C00756 V=30.0 PL=1
MOVL C00757 V=30.0 PL=1
MOVL C00758 V=30.0 PL=1
MOVL C00759 V=30.0 PL=1
MOVL C00760 V=30.0 PL=1
MOVL C00761 V=30.0 PL=1
MOVL C00762 V=30.0 PL=1
MOVL C00763 V=30.0 PL=1
MOVL C00764 V=30.0 PL=1
MOVL C00765 V=30.0 PL=1
MOVL C00766 V=30.0 PL=1
MOVL C00767 V=30.0 PL=1
MOVL C00768 V=30.0 PL=1
MOVL C00769 V=30.0 PL=1
MOVL C00770 V=30.0 PL=1
MOVL C00771 V=30.0 PL=1
MOVL C00772 V=30.0 PL=1
MOVL C00773 V=30.0 PL=1
MOVL C00774 V=30.0 PL=1
MOVL C00775 V=30.0 PL=1
MOVL C00776 V=30.0 PL=1
MOVL C00777 V=30.0 PL=1
MOVL C00778 V=30.0 PL=1
MOVL C00779 V=30.0 PL=1
MOVL C00780 V=30.0 PL=1
MOVL C00781 V=30.0 PL=1
MOVL C00782 V=30.0 PL=1
MOVL C00783 V=30.0 PL=1
MOVL C00784 V=30.0 PL=1
MOVL C00785 V=30.0 PL=1
MOVL C00786 V=30.0 PL=1
MOVL C00787 V=30.0 PL=1
MOVL C00788 V=30.0 PL=1
MOVL C00789 V=30.0 PL=1
MOVL C00790 V=30.0 PL=1
MOVL C00791 V=30.0 PL=1
MOVL C00792 V=30.0 PL=1
MOVL C00793 V=30.0 PL=1
MOVL C00794 V=30.0 PL=1
MOVL C00795 V=30.0 PL=1
MOVL C00796 V=30.0 PL=1
MOVL C00797 V=30.0 PL=1
MOVL C00798 V=30.0 PL=1
MOVL C00799 V=30.0 PL=1
MOVL C00800 V=30.0 PL=1
MOVL C00801 V=30.0 PL=1
MOVL C00802 V=30.0 PL=1
MOVL C00803 V=30.0 PL=1
MOVL C00804 V=30.0 PL=1
MOVL C00805 V=30.0 PL=1
MOVL C00806 V=30.0 PL=1
MOVL C00807 V=30.0 PL=1
MOVL C00808 V=30.0 PL=1
MOVL C00809 V=30.0 PL=1
MOVL C00810 V=30.0 PL=1
MOVL C00811 V=30.0 PL=1
MOVL C00812 V=30.0 PL=1
MOVL C00813 V=30.0 PL=1
MOVL C00814 V=30.0 PL=1
MOVL C00815 V=130.0 PL=1
MOVL C00816 V=30.0 PL=1
MOVL C00817 V=30.0 PL=1
MOVL C00818 V=30.0 PL=1
MOVL C00819 V=30.0 PL=1
MOVL C00820 V=30.0 PL=1
MOVL C00821 V=30.0 PL=1
MOVL C00822 V=30.0 PL=1
MOVL C00823 V=30.0 PL=1
MOVL C00824 V=30.0 PL=1
MOVL C00825 V=30.0 PL=1
MOVL C00826 V=30.0 PL=1
MOVL C00827 V=30.0 PL=1
MOVL C00828 V=30.0 PL=1
MOVL C00829 V=30.0 PL=1
MOVL C00830 V=30.0 PL=1
MOVL C00831 V=30.0 PL=1
MOVL C00832 V=30.0 PL=1
MOVL C00833 V=30.0 PL=1
MOVL C00834 V=30.0 PL=1
MOVL C00835 V=30.0 PL=1
MOVL C00836 V=30.0 PL=1
MOVL C00837 V=30.0 PL=1
MOVL C00838 V=30.0 PL=1
MOVL C00839 V=30.0 PL=1
MOVL C00840 V=30.0 PL=1
MOVL C00841 V=30.0 PL=1
MOVL C00842 V=30.0 PL=1
MOVL C00843 V=30.0 PL=1
MOVL C00844 V=30.0 PL=1
MOVL C00845 V=30.0 PL=1
MOVL C00846 V=30.0 PL=1
MOVL C00847 V=30.0 PL=1
MOVL C00848 V=30.0 PL=1
MOVL C00849 V=30.0 PL=1
MOVL C00850 V=30.0 PL=1
MOVL C00851 V=30.0 PL=1
MOVL C00852 V=30.0 PL=1
MOVL C00853 V=30.0 PL=1
MOVL C00854 V=30.0 PL=1
MOVL C00855 V=30.0 PL=1
MOVL C00856 V=30.0 PL=1
MOVL C00857 V=30.0 PL=1
MOVL C00858 V=30.0 PL=1
MOVL C00859 V=30.0 PL=1
MOVL C00860 V=30.0 PL=1
MOVL C00861 V=30.0 PL=1
MOVL C00862 V=30.0 PL=1
MOVL C00863 V=30.0 PL=1
MOVL C00864 V=30.0 PL=1
MOVL C00865 V=30.0 PL=1
MOVL C00866 V=30.0 PL=1
MOVL C00867 V=30.0 PL=1
MOVL C00868 V=30.0 PL=1
MOVL C00869 V=30.0 PL=1
MOVL C00870 V=30.0 PL=1
MOVL C00871 V=30.0 PL=1
MOVL C00872 V=30.0 PL=1
MOVL C00873 V=30.0 PL=1
MOVL C00874 V=30.0 PL=1
MOVL C00875 V=30.0 PL=1
MOVL C00876 V=30.0 PL=1
MOVL C00877 V=30.0 PL=1
MOVL C00878 V=30.0 PL=1
MOVL C00879 V=30.0 PL=1
MOVL C00880 V=30.0 PL=1
MOVL C00881 V=30.0 PL=1
MOVL C00882 V=30.0 PL=1
MOVL C00883 V=30.0 PL=1
MOVL C00884 V=30.0 PL=1
MOVL C00885 V=30.0 PL=1
MOVL C00886 V=30.0 PL=1
MOVL C00887 V=30.0 PL=1
MOVL C00888 V=30.0 PL=1
MOVL C00889 V=30.0 PL=1
MOVL C00890 V=30.0 PL=1
MOVL C00891 V=30.0 PL=1
MOVL C00892 V=30.0 PL=1
MOVL C00893 V=30.0 PL=1
MOVL C00894 V=30.0 PL=1
MOVL C00895 V=30.0 PL=1
MOVL C00896 V=30.0 PL=1
MOVL C00897 V=30.0 PL=1
MOVL C00898 V=30.0 PL=1
MOVL C00899 V=30.0 PL=1
MOVL C00900 V=30.0 PL=1
MOVL C00901 V=30.0 PL=1
MOVL C00902 V=30.0 PL=1
MOVL C00903 V=30.0 PL=1
MOVL C00904 V=130.0 PL=1
MOVL C00905 V=80.0 PL=1
MOVL C00906 V=130.0 PL=1
MOVL C00907 V=80.0 PL=1
MOVL C00908 V=130.0 PL=1
MOVL C00909 V=80.0 PL=1
MOVL C00910 V=130.0 PL=1
MOVL C00911 V=80.0 PL=1
MOVL C00912 V=80.0 PL=1
MOVL C00913 V=80.0 PL=1
MOVL C00914 V=80.0 PL=1
MOVL C00915 V=80.0 PL=1
MOVL C00916 V=80.0 PL=1
MOVL C00917 V=80.0 PL=1
MOVL C00918 V=80.0 PL=1
MOVL C00919 V=80.0 PL=1
MOVL C00920 V=80.0 PL=1
MOVL C00921 V=80.0 PL=1
MOVL C00922 V=80.0 PL=1
MOVL C00923 V=80.0 PL=1
MOVL C00924 V=130.0 PL=1
MOVL C00925 V=130.0 PL=1
MOVL C00926 V=60.0 PL=1
MOVL C00927 V=60.0 PL=1
MOVL C00928 V=60.0 PL=1
MOVL C00929 V=60.0 PL=1
MOVL C00930 V=60.0 PL=1
MOVL C00931 V=60.0 PL=1
MOVL C00932 V=60.0 PL=1
MOVL C00933 V=60.0 PL=1
MOVL C00934 V=60.0 PL=1
MOVL C00935 V=60.0 PL=1
MOVL C00936 V=60.0 PL=1
MOVL C00937 V=60.0 PL=1
MOVL C00938 V=60.0 PL=1
MOVL C00939 V=60.0 PL=1
MOVL C00940 V=60.0 PL=1
MOVL C00941 V=60.0 PL=1
MOVL C00942 V=60.0 PL=1
MOVL C00943 V=60.0 PL=1
MOVL C00944 V=60.0 PL=1
MOVL C00945 V=60.0 PL=1
MOVL C00946 V=60.0 PL=1
MOVL C00947 V=60.0 PL=1
MOVL C00948 V=60.0 PL=1
MOVL C00949 V=60.0 PL=1
MOVL C00950 V=130.0 PL=1
MOVL C00951 V=60.0 PL=1
MOVL C00952 V=60.0 PL=1
MOVL C00953 V=60.0 PL=1
MOVL C00954 V=60.0 PL=1
MOVL C00955 V=60.0 PL=1
MOVL C00956 V=60.0 PL=1
MOVL C00957 V=60.0 PL=1
MOVL C00958 V=60.0 PL=1
MOVL C00959 V=60.0 PL=1
MOVL C00960 V=60.0 PL=1
MOVL C00961 V=60.0 PL=1
MOVL C00962 V=60.0 PL=1
MOVL C00963 V=60.0 PL=1
MOVL C00964 V=60.0 PL=1
MOVL C00965 V=60.0 PL=1
MOVL C00966 V=60.0 PL=1
MOVL C00967 V=60.0 PL=1
MOVL C00968 V=60.0 PL=1
MOVL C00969 V=60.0 PL=1
MOVL C00970 V=60.0 PL=1
MOVL C00971 V=60.0 PL=1
MOVL C00972 V=60.0 PL=1
MOVL C00973 V=60.0 PL=1
MOVL C00974 V=60.0 PL=1
MOVL C00975 V=60.0 PL=1
MOVL C00976 V=60.0 PL=1
MOVL C00977 V=60.0 PL=1
MOVL C00978 V=60.0 PL=1
MOVL C00979 V=60.0 PL=1
MOVL C00980 V=60.0 PL=1
MOVL C00981 V=60.0 PL=1
MOVL C00982 V=60.0 PL=1
MOVL C00983 V=60.0 PL=1
MOVL C00984 V=60.0 PL=1
MOVL C00985 V=60.0 PL=1
MOVL C00986 V=60.0 PL=1
MOVL C00987 V=60.0 PL=1
MOVL C00988 V=60.0 PL=1
MOVL C00989 V=60.0 PL=1
MOVL C00990 V=60.0 PL=1
MOVL C00991 V=60.0 PL=1
MOVL C00992 V=60.0 PL=1
MOVL C00993 V=130.0 PL=1
MOVL C00994 V=30.0 PL=1
MOVL C00995 V=30.0 PL=1
MOVL C00996 V=30.0 PL=1
MOVL C00997 V=30.0 PL=1
MOVL C00998 V=30.0 PL=1
MOVL C00999 V=30.0 PL=1
MOVL C01000 V=30.0 PL=1
MOVL C01001 V=30.0 PL=1
MOVL C01002 V=30.0 PL=1
END
